   // GBK_TO_UNICODE[19568] := 16#BBEA;
   // GBK_TO_UNICODE[19569] := 16#9B42;
   // GBK_TO_UNICODE[19570] := 16#BBEB;
   // GBK_TO_UNICODE[19571] := 16#6D51;
   // GBK_TO_UNICODE[19572] := 16#BBEC;
   // GBK_TO_UNICODE[19573] := 16#6DF7;
   // GBK_TO_UNICODE[19574] := 16#BBED;
   // GBK_TO_UNICODE[19575] := 16#8C41;
   // GBK_TO_UNICODE[19576] := 16#BBEE;
   // GBK_TO_UNICODE[19577] := 16#6D3B;
   // GBK_TO_UNICODE[19578] := 16#BBEF;
   // GBK_TO_UNICODE[19579] := 16#4F19;
   // GBK_TO_UNICODE[19580] := 16#BBF0;
   // GBK_TO_UNICODE[19581] := 16#706B;
   // GBK_TO_UNICODE[19582] := 16#BBF1;
   // GBK_TO_UNICODE[19583] := 16#83B7;
   // GBK_TO_UNICODE[19584] := 16#BBF2;
   // GBK_TO_UNICODE[19585] := 16#6216;
   // GBK_TO_UNICODE[19586] := 16#BBF3;
   // GBK_TO_UNICODE[19587] := 16#60D1;
   // GBK_TO_UNICODE[19588] := 16#BBF4;
   // GBK_TO_UNICODE[19589] := 16#970D;
   // GBK_TO_UNICODE[19590] := 16#BBF5;
   // GBK_TO_UNICODE[19591] := 16#8D27;
   // GBK_TO_UNICODE[19592] := 16#BBF6;
   // GBK_TO_UNICODE[19593] := 16#7978;
   // GBK_TO_UNICODE[19594] := 16#BBF7;
   // GBK_TO_UNICODE[19595] := 16#51FB;
   // GBK_TO_UNICODE[19596] := 16#BBF8;
   // GBK_TO_UNICODE[19597] := 16#573E;
   // GBK_TO_UNICODE[19598] := 16#BBF9;
   // GBK_TO_UNICODE[19599] := 16#57FA;
   // GBK_TO_UNICODE[19600] := 16#BBFA;
   // GBK_TO_UNICODE[19601] := 16#673A;
   // GBK_TO_UNICODE[19602] := 16#BBFB;
   // GBK_TO_UNICODE[19603] := 16#7578;
   // GBK_TO_UNICODE[19604] := 16#BBFC;
   // GBK_TO_UNICODE[19605] := 16#7A3D;
   // GBK_TO_UNICODE[19606] := 16#BBFD;
   // GBK_TO_UNICODE[19607] := 16#79EF;
   // GBK_TO_UNICODE[19608] := 16#BBFE;
   // GBK_TO_UNICODE[19609] := 16#7B95;
   // GBK_TO_UNICODE[19610] := 16#BC40;
   // GBK_TO_UNICODE[19611] := 16#7CBF;
   // GBK_TO_UNICODE[19612] := 16#BC41;
   // GBK_TO_UNICODE[19613] := 16#7CC0;
   // GBK_TO_UNICODE[19614] := 16#BC42;
   // GBK_TO_UNICODE[19615] := 16#7CC2;
   // GBK_TO_UNICODE[19616] := 16#BC43;
   // GBK_TO_UNICODE[19617] := 16#7CC3;
   // GBK_TO_UNICODE[19618] := 16#BC44;
   // GBK_TO_UNICODE[19619] := 16#7CC4;
   // GBK_TO_UNICODE[19620] := 16#BC45;
   // GBK_TO_UNICODE[19621] := 16#7CC6;
   // GBK_TO_UNICODE[19622] := 16#BC46;
   // GBK_TO_UNICODE[19623] := 16#7CC9;
   // GBK_TO_UNICODE[19624] := 16#BC47;
   // GBK_TO_UNICODE[19625] := 16#7CCB;
   // GBK_TO_UNICODE[19626] := 16#BC48;
   // GBK_TO_UNICODE[19627] := 16#7CCE;
   // GBK_TO_UNICODE[19628] := 16#BC49;
   // GBK_TO_UNICODE[19629] := 16#7CCF;
   // GBK_TO_UNICODE[19630] := 16#BC4A;
   // GBK_TO_UNICODE[19631] := 16#7CD0;
   // GBK_TO_UNICODE[19632] := 16#BC4B;
   // GBK_TO_UNICODE[19633] := 16#7CD1;
   // GBK_TO_UNICODE[19634] := 16#BC4C;
   // GBK_TO_UNICODE[19635] := 16#7CD2;
   // GBK_TO_UNICODE[19636] := 16#BC4D;
   // GBK_TO_UNICODE[19637] := 16#7CD3;
   // GBK_TO_UNICODE[19638] := 16#BC4E;
   // GBK_TO_UNICODE[19639] := 16#7CD4;
   // GBK_TO_UNICODE[19640] := 16#BC4F;
   // GBK_TO_UNICODE[19641] := 16#7CD8;
   // GBK_TO_UNICODE[19642] := 16#BC50;
   // GBK_TO_UNICODE[19643] := 16#7CDA;
   // GBK_TO_UNICODE[19644] := 16#BC51;
   // GBK_TO_UNICODE[19645] := 16#7CDB;
   // GBK_TO_UNICODE[19646] := 16#BC52;
   // GBK_TO_UNICODE[19647] := 16#7CDD;
   // GBK_TO_UNICODE[19648] := 16#BC53;
   // GBK_TO_UNICODE[19649] := 16#7CDE;
   // GBK_TO_UNICODE[19650] := 16#BC54;
   // GBK_TO_UNICODE[19651] := 16#7CE1;
   // GBK_TO_UNICODE[19652] := 16#BC55;
   // GBK_TO_UNICODE[19653] := 16#7CE2;
   // GBK_TO_UNICODE[19654] := 16#BC56;
   // GBK_TO_UNICODE[19655] := 16#7CE3;
   // GBK_TO_UNICODE[19656] := 16#BC57;
   // GBK_TO_UNICODE[19657] := 16#7CE4;
   // GBK_TO_UNICODE[19658] := 16#BC58;
   // GBK_TO_UNICODE[19659] := 16#7CE5;
   // GBK_TO_UNICODE[19660] := 16#BC59;
   // GBK_TO_UNICODE[19661] := 16#7CE6;
   // GBK_TO_UNICODE[19662] := 16#BC5A;
   // GBK_TO_UNICODE[19663] := 16#7CE7;
   // GBK_TO_UNICODE[19664] := 16#BC5B;
   // GBK_TO_UNICODE[19665] := 16#7CE9;
   // GBK_TO_UNICODE[19666] := 16#BC5C;
   // GBK_TO_UNICODE[19667] := 16#7CEA;
   // GBK_TO_UNICODE[19668] := 16#BC5D;
   // GBK_TO_UNICODE[19669] := 16#7CEB;
   // GBK_TO_UNICODE[19670] := 16#BC5E;
   // GBK_TO_UNICODE[19671] := 16#7CEC;
   // GBK_TO_UNICODE[19672] := 16#BC5F;
   // GBK_TO_UNICODE[19673] := 16#7CED;
   // GBK_TO_UNICODE[19674] := 16#BC60;
   // GBK_TO_UNICODE[19675] := 16#7CEE;
   // GBK_TO_UNICODE[19676] := 16#BC61;
   // GBK_TO_UNICODE[19677] := 16#7CF0;
   // GBK_TO_UNICODE[19678] := 16#BC62;
   // GBK_TO_UNICODE[19679] := 16#7CF1;
   // GBK_TO_UNICODE[19680] := 16#BC63;
   // GBK_TO_UNICODE[19681] := 16#7CF2;
   // GBK_TO_UNICODE[19682] := 16#BC64;
   // GBK_TO_UNICODE[19683] := 16#7CF3;
   // GBK_TO_UNICODE[19684] := 16#BC65;
   // GBK_TO_UNICODE[19685] := 16#7CF4;
   // GBK_TO_UNICODE[19686] := 16#BC66;
   // GBK_TO_UNICODE[19687] := 16#7CF5;
   // GBK_TO_UNICODE[19688] := 16#BC67;
   // GBK_TO_UNICODE[19689] := 16#7CF6;
   // GBK_TO_UNICODE[19690] := 16#BC68;
   // GBK_TO_UNICODE[19691] := 16#7CF7;
   // GBK_TO_UNICODE[19692] := 16#BC69;
   // GBK_TO_UNICODE[19693] := 16#7CF9;
   // GBK_TO_UNICODE[19694] := 16#BC6A;
   // GBK_TO_UNICODE[19695] := 16#7CFA;
   // GBK_TO_UNICODE[19696] := 16#BC6B;
   // GBK_TO_UNICODE[19697] := 16#7CFC;
   // GBK_TO_UNICODE[19698] := 16#BC6C;
   // GBK_TO_UNICODE[19699] := 16#7CFD;
   // GBK_TO_UNICODE[19700] := 16#BC6D;
   // GBK_TO_UNICODE[19701] := 16#7CFE;
   // GBK_TO_UNICODE[19702] := 16#BC6E;
   // GBK_TO_UNICODE[19703] := 16#7CFF;
   // GBK_TO_UNICODE[19704] := 16#BC6F;
   // GBK_TO_UNICODE[19705] := 16#7D00;
   // GBK_TO_UNICODE[19706] := 16#BC70;
   // GBK_TO_UNICODE[19707] := 16#7D01;
   // GBK_TO_UNICODE[19708] := 16#BC71;
   // GBK_TO_UNICODE[19709] := 16#7D02;
   // GBK_TO_UNICODE[19710] := 16#BC72;
   // GBK_TO_UNICODE[19711] := 16#7D03;
   // GBK_TO_UNICODE[19712] := 16#BC73;
   // GBK_TO_UNICODE[19713] := 16#7D04;
   // GBK_TO_UNICODE[19714] := 16#BC74;
   // GBK_TO_UNICODE[19715] := 16#7D05;
   // GBK_TO_UNICODE[19716] := 16#BC75;
   // GBK_TO_UNICODE[19717] := 16#7D06;
   // GBK_TO_UNICODE[19718] := 16#BC76;
   // GBK_TO_UNICODE[19719] := 16#7D07;
   // GBK_TO_UNICODE[19720] := 16#BC77;
   // GBK_TO_UNICODE[19721] := 16#7D08;
   // GBK_TO_UNICODE[19722] := 16#BC78;
   // GBK_TO_UNICODE[19723] := 16#7D09;
   // GBK_TO_UNICODE[19724] := 16#BC79;
   // GBK_TO_UNICODE[19725] := 16#7D0B;
   // GBK_TO_UNICODE[19726] := 16#BC7A;
   // GBK_TO_UNICODE[19727] := 16#7D0C;
   // GBK_TO_UNICODE[19728] := 16#BC7B;
   // GBK_TO_UNICODE[19729] := 16#7D0D;
   // GBK_TO_UNICODE[19730] := 16#BC7C;
   // GBK_TO_UNICODE[19731] := 16#7D0E;
   // GBK_TO_UNICODE[19732] := 16#BC7D;
   // GBK_TO_UNICODE[19733] := 16#7D0F;
   // GBK_TO_UNICODE[19734] := 16#BC7E;
   // GBK_TO_UNICODE[19735] := 16#7D10;
   // GBK_TO_UNICODE[19736] := 16#BC80;
   // GBK_TO_UNICODE[19737] := 16#7D11;
   // GBK_TO_UNICODE[19738] := 16#BC81;
   // GBK_TO_UNICODE[19739] := 16#7D12;
   // GBK_TO_UNICODE[19740] := 16#BC82;
   // GBK_TO_UNICODE[19741] := 16#7D13;
   // GBK_TO_UNICODE[19742] := 16#BC83;
   // GBK_TO_UNICODE[19743] := 16#7D14;
   // GBK_TO_UNICODE[19744] := 16#BC84;
   // GBK_TO_UNICODE[19745] := 16#7D15;
   // GBK_TO_UNICODE[19746] := 16#BC85;
   // GBK_TO_UNICODE[19747] := 16#7D16;
   // GBK_TO_UNICODE[19748] := 16#BC86;
   // GBK_TO_UNICODE[19749] := 16#7D17;
   // GBK_TO_UNICODE[19750] := 16#BC87;
   // GBK_TO_UNICODE[19751] := 16#7D18;
   // GBK_TO_UNICODE[19752] := 16#BC88;
   // GBK_TO_UNICODE[19753] := 16#7D19;
   // GBK_TO_UNICODE[19754] := 16#BC89;
   // GBK_TO_UNICODE[19755] := 16#7D1A;
   // GBK_TO_UNICODE[19756] := 16#BC8A;
   // GBK_TO_UNICODE[19757] := 16#7D1B;
   // GBK_TO_UNICODE[19758] := 16#BC8B;
   // GBK_TO_UNICODE[19759] := 16#7D1C;
   // GBK_TO_UNICODE[19760] := 16#BC8C;
   // GBK_TO_UNICODE[19761] := 16#7D1D;
   // GBK_TO_UNICODE[19762] := 16#BC8D;
   // GBK_TO_UNICODE[19763] := 16#7D1E;
   // GBK_TO_UNICODE[19764] := 16#BC8E;
   // GBK_TO_UNICODE[19765] := 16#7D1F;
   // GBK_TO_UNICODE[19766] := 16#BC8F;
   // GBK_TO_UNICODE[19767] := 16#7D21;
   // GBK_TO_UNICODE[19768] := 16#BC90;
   // GBK_TO_UNICODE[19769] := 16#7D23;
   // GBK_TO_UNICODE[19770] := 16#BC91;
   // GBK_TO_UNICODE[19771] := 16#7D24;
   // GBK_TO_UNICODE[19772] := 16#BC92;
   // GBK_TO_UNICODE[19773] := 16#7D25;
   // GBK_TO_UNICODE[19774] := 16#BC93;
   // GBK_TO_UNICODE[19775] := 16#7D26;
   // GBK_TO_UNICODE[19776] := 16#BC94;
   // GBK_TO_UNICODE[19777] := 16#7D28;
   // GBK_TO_UNICODE[19778] := 16#BC95;
   // GBK_TO_UNICODE[19779] := 16#7D29;
   // GBK_TO_UNICODE[19780] := 16#BC96;
   // GBK_TO_UNICODE[19781] := 16#7D2A;
   // GBK_TO_UNICODE[19782] := 16#BC97;
   // GBK_TO_UNICODE[19783] := 16#7D2C;
   // GBK_TO_UNICODE[19784] := 16#BC98;
   // GBK_TO_UNICODE[19785] := 16#7D2D;
   // GBK_TO_UNICODE[19786] := 16#BC99;
   // GBK_TO_UNICODE[19787] := 16#7D2E;
   // GBK_TO_UNICODE[19788] := 16#BC9A;
   // GBK_TO_UNICODE[19789] := 16#7D30;
   // GBK_TO_UNICODE[19790] := 16#BC9B;
   // GBK_TO_UNICODE[19791] := 16#7D31;
   // GBK_TO_UNICODE[19792] := 16#BC9C;
   // GBK_TO_UNICODE[19793] := 16#7D32;
   // GBK_TO_UNICODE[19794] := 16#BC9D;
   // GBK_TO_UNICODE[19795] := 16#7D33;
   // GBK_TO_UNICODE[19796] := 16#BC9E;
   // GBK_TO_UNICODE[19797] := 16#7D34;
   // GBK_TO_UNICODE[19798] := 16#BC9F;
   // GBK_TO_UNICODE[19799] := 16#7D35;
   // GBK_TO_UNICODE[19800] := 16#BCA0;
   // GBK_TO_UNICODE[19801] := 16#7D36;
   // GBK_TO_UNICODE[19802] := 16#BCA1;
   // GBK_TO_UNICODE[19803] := 16#808C;
   // GBK_TO_UNICODE[19804] := 16#BCA2;
   // GBK_TO_UNICODE[19805] := 16#9965;
   // GBK_TO_UNICODE[19806] := 16#BCA3;
   // GBK_TO_UNICODE[19807] := 16#8FF9;
   // GBK_TO_UNICODE[19808] := 16#BCA4;
   // GBK_TO_UNICODE[19809] := 16#6FC0;
   // GBK_TO_UNICODE[19810] := 16#BCA5;
   // GBK_TO_UNICODE[19811] := 16#8BA5;
   // GBK_TO_UNICODE[19812] := 16#BCA6;
   // GBK_TO_UNICODE[19813] := 16#9E21;
   // GBK_TO_UNICODE[19814] := 16#BCA7;
   // GBK_TO_UNICODE[19815] := 16#59EC;
   // GBK_TO_UNICODE[19816] := 16#BCA8;
   // GBK_TO_UNICODE[19817] := 16#7EE9;
   // GBK_TO_UNICODE[19818] := 16#BCA9;
   // GBK_TO_UNICODE[19819] := 16#7F09;
   // GBK_TO_UNICODE[19820] := 16#BCAA;
   // GBK_TO_UNICODE[19821] := 16#5409;
   // GBK_TO_UNICODE[19822] := 16#BCAB;
   // GBK_TO_UNICODE[19823] := 16#6781;
   // GBK_TO_UNICODE[19824] := 16#BCAC;
   // GBK_TO_UNICODE[19825] := 16#68D8;
   // GBK_TO_UNICODE[19826] := 16#BCAD;
   // GBK_TO_UNICODE[19827] := 16#8F91;
   // GBK_TO_UNICODE[19828] := 16#BCAE;
   // GBK_TO_UNICODE[19829] := 16#7C4D;
   // GBK_TO_UNICODE[19830] := 16#BCAF;
   // GBK_TO_UNICODE[19831] := 16#96C6;
   // GBK_TO_UNICODE[19832] := 16#BCB0;
   // GBK_TO_UNICODE[19833] := 16#53CA;
   // GBK_TO_UNICODE[19834] := 16#BCB1;
   // GBK_TO_UNICODE[19835] := 16#6025;
   // GBK_TO_UNICODE[19836] := 16#BCB2;
   // GBK_TO_UNICODE[19837] := 16#75BE;
   // GBK_TO_UNICODE[19838] := 16#BCB3;
   // GBK_TO_UNICODE[19839] := 16#6C72;
   // GBK_TO_UNICODE[19840] := 16#BCB4;
   // GBK_TO_UNICODE[19841] := 16#5373;
   // GBK_TO_UNICODE[19842] := 16#BCB5;
   // GBK_TO_UNICODE[19843] := 16#5AC9;
   // GBK_TO_UNICODE[19844] := 16#BCB6;
   // GBK_TO_UNICODE[19845] := 16#7EA7;
   // GBK_TO_UNICODE[19846] := 16#BCB7;
   // GBK_TO_UNICODE[19847] := 16#6324;
   // GBK_TO_UNICODE[19848] := 16#BCB8;
   // GBK_TO_UNICODE[19849] := 16#51E0;
   // GBK_TO_UNICODE[19850] := 16#BCB9;
   // GBK_TO_UNICODE[19851] := 16#810A;
   // GBK_TO_UNICODE[19852] := 16#BCBA;
   // GBK_TO_UNICODE[19853] := 16#5DF1;
   // GBK_TO_UNICODE[19854] := 16#BCBB;
   // GBK_TO_UNICODE[19855] := 16#84DF;
   // GBK_TO_UNICODE[19856] := 16#BCBC;
   // GBK_TO_UNICODE[19857] := 16#6280;
   // GBK_TO_UNICODE[19858] := 16#BCBD;
   // GBK_TO_UNICODE[19859] := 16#5180;
   // GBK_TO_UNICODE[19860] := 16#BCBE;
   // GBK_TO_UNICODE[19861] := 16#5B63;
   // GBK_TO_UNICODE[19862] := 16#BCBF;
   // GBK_TO_UNICODE[19863] := 16#4F0E;
   // GBK_TO_UNICODE[19864] := 16#BCC0;
   // GBK_TO_UNICODE[19865] := 16#796D;
   // GBK_TO_UNICODE[19866] := 16#BCC1;
   // GBK_TO_UNICODE[19867] := 16#5242;
   // GBK_TO_UNICODE[19868] := 16#BCC2;
   // GBK_TO_UNICODE[19869] := 16#60B8;
   // GBK_TO_UNICODE[19870] := 16#BCC3;
   // GBK_TO_UNICODE[19871] := 16#6D4E;
   // GBK_TO_UNICODE[19872] := 16#BCC4;
   // GBK_TO_UNICODE[19873] := 16#5BC4;
   // GBK_TO_UNICODE[19874] := 16#BCC5;
   // GBK_TO_UNICODE[19875] := 16#5BC2;
   // GBK_TO_UNICODE[19876] := 16#BCC6;
   // GBK_TO_UNICODE[19877] := 16#8BA1;
   // GBK_TO_UNICODE[19878] := 16#BCC7;
   // GBK_TO_UNICODE[19879] := 16#8BB0;
   // GBK_TO_UNICODE[19880] := 16#BCC8;
   // GBK_TO_UNICODE[19881] := 16#65E2;
   // GBK_TO_UNICODE[19882] := 16#BCC9;
   // GBK_TO_UNICODE[19883] := 16#5FCC;
   // GBK_TO_UNICODE[19884] := 16#BCCA;
   // GBK_TO_UNICODE[19885] := 16#9645;
   // GBK_TO_UNICODE[19886] := 16#BCCB;
   // GBK_TO_UNICODE[19887] := 16#5993;
   // GBK_TO_UNICODE[19888] := 16#BCCC;
   // GBK_TO_UNICODE[19889] := 16#7EE7;
   // GBK_TO_UNICODE[19890] := 16#BCCD;
   // GBK_TO_UNICODE[19891] := 16#7EAA;
   // GBK_TO_UNICODE[19892] := 16#BCCE;
   // GBK_TO_UNICODE[19893] := 16#5609;
   // GBK_TO_UNICODE[19894] := 16#BCCF;
   // GBK_TO_UNICODE[19895] := 16#67B7;
   // GBK_TO_UNICODE[19896] := 16#BCD0;
   // GBK_TO_UNICODE[19897] := 16#5939;
   // GBK_TO_UNICODE[19898] := 16#BCD1;
   // GBK_TO_UNICODE[19899] := 16#4F73;
   // GBK_TO_UNICODE[19900] := 16#BCD2;
   // GBK_TO_UNICODE[19901] := 16#5BB6;
   // GBK_TO_UNICODE[19902] := 16#BCD3;
   // GBK_TO_UNICODE[19903] := 16#52A0;
   // GBK_TO_UNICODE[19904] := 16#BCD4;
   // GBK_TO_UNICODE[19905] := 16#835A;
   // GBK_TO_UNICODE[19906] := 16#BCD5;
   // GBK_TO_UNICODE[19907] := 16#988A;
   // GBK_TO_UNICODE[19908] := 16#BCD6;
   // GBK_TO_UNICODE[19909] := 16#8D3E;
   // GBK_TO_UNICODE[19910] := 16#BCD7;
   // GBK_TO_UNICODE[19911] := 16#7532;
   // GBK_TO_UNICODE[19912] := 16#BCD8;
   // GBK_TO_UNICODE[19913] := 16#94BE;
   // GBK_TO_UNICODE[19914] := 16#BCD9;
   // GBK_TO_UNICODE[19915] := 16#5047;
   // GBK_TO_UNICODE[19916] := 16#BCDA;
   // GBK_TO_UNICODE[19917] := 16#7A3C;
   // GBK_TO_UNICODE[19918] := 16#BCDB;
   // GBK_TO_UNICODE[19919] := 16#4EF7;
   // GBK_TO_UNICODE[19920] := 16#BCDC;
   // GBK_TO_UNICODE[19921] := 16#67B6;
   // GBK_TO_UNICODE[19922] := 16#BCDD;
   // GBK_TO_UNICODE[19923] := 16#9A7E;
   // GBK_TO_UNICODE[19924] := 16#BCDE;
   // GBK_TO_UNICODE[19925] := 16#5AC1;
   // GBK_TO_UNICODE[19926] := 16#BCDF;
   // GBK_TO_UNICODE[19927] := 16#6B7C;
   // GBK_TO_UNICODE[19928] := 16#BCE0;
   // GBK_TO_UNICODE[19929] := 16#76D1;
   // GBK_TO_UNICODE[19930] := 16#BCE1;
   // GBK_TO_UNICODE[19931] := 16#575A;
   // GBK_TO_UNICODE[19932] := 16#BCE2;
   // GBK_TO_UNICODE[19933] := 16#5C16;
   // GBK_TO_UNICODE[19934] := 16#BCE3;
   // GBK_TO_UNICODE[19935] := 16#7B3A;
   // GBK_TO_UNICODE[19936] := 16#BCE4;
   // GBK_TO_UNICODE[19937] := 16#95F4;
   // GBK_TO_UNICODE[19938] := 16#BCE5;
   // GBK_TO_UNICODE[19939] := 16#714E;
   // GBK_TO_UNICODE[19940] := 16#BCE6;
   // GBK_TO_UNICODE[19941] := 16#517C;
   // GBK_TO_UNICODE[19942] := 16#BCE7;
   // GBK_TO_UNICODE[19943] := 16#80A9;
   // GBK_TO_UNICODE[19944] := 16#BCE8;
   // GBK_TO_UNICODE[19945] := 16#8270;
   // GBK_TO_UNICODE[19946] := 16#BCE9;
   // GBK_TO_UNICODE[19947] := 16#5978;
   // GBK_TO_UNICODE[19948] := 16#BCEA;
   // GBK_TO_UNICODE[19949] := 16#7F04;
   // GBK_TO_UNICODE[19950] := 16#BCEB;
   // GBK_TO_UNICODE[19951] := 16#8327;
   // GBK_TO_UNICODE[19952] := 16#BCEC;
   // GBK_TO_UNICODE[19953] := 16#68C0;
   // GBK_TO_UNICODE[19954] := 16#BCED;
   // GBK_TO_UNICODE[19955] := 16#67EC;
   // GBK_TO_UNICODE[19956] := 16#BCEE;
   // GBK_TO_UNICODE[19957] := 16#78B1;
   // GBK_TO_UNICODE[19958] := 16#BCEF;
   // GBK_TO_UNICODE[19959] := 16#7877;
   // GBK_TO_UNICODE[19960] := 16#BCF0;
   // GBK_TO_UNICODE[19961] := 16#62E3;
   // GBK_TO_UNICODE[19962] := 16#BCF1;
   // GBK_TO_UNICODE[19963] := 16#6361;
   // GBK_TO_UNICODE[19964] := 16#BCF2;
   // GBK_TO_UNICODE[19965] := 16#7B80;
   // GBK_TO_UNICODE[19966] := 16#BCF3;
   // GBK_TO_UNICODE[19967] := 16#4FED;
   // GBK_TO_UNICODE[19968] := 16#BCF4;
   // GBK_TO_UNICODE[19969] := 16#526A;
   // GBK_TO_UNICODE[19970] := 16#BCF5;
   // GBK_TO_UNICODE[19971] := 16#51CF;
   // GBK_TO_UNICODE[19972] := 16#BCF6;
   // GBK_TO_UNICODE[19973] := 16#8350;
   // GBK_TO_UNICODE[19974] := 16#BCF7;
   // GBK_TO_UNICODE[19975] := 16#69DB;
   // GBK_TO_UNICODE[19976] := 16#BCF8;
   // GBK_TO_UNICODE[19977] := 16#9274;
   // GBK_TO_UNICODE[19978] := 16#BCF9;
   // GBK_TO_UNICODE[19979] := 16#8DF5;
   // GBK_TO_UNICODE[19980] := 16#BCFA;
   // GBK_TO_UNICODE[19981] := 16#8D31;
   // GBK_TO_UNICODE[19982] := 16#BCFB;
   // GBK_TO_UNICODE[19983] := 16#89C1;
   // GBK_TO_UNICODE[19984] := 16#BCFC;
   // GBK_TO_UNICODE[19985] := 16#952E;
   // GBK_TO_UNICODE[19986] := 16#BCFD;
   // GBK_TO_UNICODE[19987] := 16#7BAD;
   // GBK_TO_UNICODE[19988] := 16#BCFE;
   // GBK_TO_UNICODE[19989] := 16#4EF6;
   // GBK_TO_UNICODE[19990] := 16#BD40;
   // GBK_TO_UNICODE[19991] := 16#7D37;
   // GBK_TO_UNICODE[19992] := 16#BD41;
   // GBK_TO_UNICODE[19993] := 16#7D38;
   // GBK_TO_UNICODE[19994] := 16#BD42;
   // GBK_TO_UNICODE[19995] := 16#7D39;
   // GBK_TO_UNICODE[19996] := 16#BD43;
   // GBK_TO_UNICODE[19997] := 16#7D3A;
   // GBK_TO_UNICODE[19998] := 16#BD44;
   // GBK_TO_UNICODE[19999] := 16#7D3B;
   // GBK_TO_UNICODE[20000] := 16#BD45;
   // GBK_TO_UNICODE[20001] := 16#7D3C;
   // GBK_TO_UNICODE[20002] := 16#BD46;
   // GBK_TO_UNICODE[20003] := 16#7D3D;
   // GBK_TO_UNICODE[20004] := 16#BD47;
   // GBK_TO_UNICODE[20005] := 16#7D3E;
   // GBK_TO_UNICODE[20006] := 16#BD48;
   // GBK_TO_UNICODE[20007] := 16#7D3F;
   // GBK_TO_UNICODE[20008] := 16#BD49;
   // GBK_TO_UNICODE[20009] := 16#7D40;
   // GBK_TO_UNICODE[20010] := 16#BD4A;
   // GBK_TO_UNICODE[20011] := 16#7D41;
   // GBK_TO_UNICODE[20012] := 16#BD4B;
   // GBK_TO_UNICODE[20013] := 16#7D42;
   // GBK_TO_UNICODE[20014] := 16#BD4C;
   // GBK_TO_UNICODE[20015] := 16#7D43;
   // GBK_TO_UNICODE[20016] := 16#BD4D;
   // GBK_TO_UNICODE[20017] := 16#7D44;
   // GBK_TO_UNICODE[20018] := 16#BD4E;
   // GBK_TO_UNICODE[20019] := 16#7D45;
   // GBK_TO_UNICODE[20020] := 16#BD4F;
   // GBK_TO_UNICODE[20021] := 16#7D46;
   // GBK_TO_UNICODE[20022] := 16#BD50;
   // GBK_TO_UNICODE[20023] := 16#7D47;
   // GBK_TO_UNICODE[20024] := 16#BD51;
   // GBK_TO_UNICODE[20025] := 16#7D48;
   // GBK_TO_UNICODE[20026] := 16#BD52;
   // GBK_TO_UNICODE[20027] := 16#7D49;
   // GBK_TO_UNICODE[20028] := 16#BD53;
   // GBK_TO_UNICODE[20029] := 16#7D4A;
   // GBK_TO_UNICODE[20030] := 16#BD54;
   // GBK_TO_UNICODE[20031] := 16#7D4B;
   // GBK_TO_UNICODE[20032] := 16#BD55;
   // GBK_TO_UNICODE[20033] := 16#7D4C;
   // GBK_TO_UNICODE[20034] := 16#BD56;
   // GBK_TO_UNICODE[20035] := 16#7D4D;
   // GBK_TO_UNICODE[20036] := 16#BD57;
   // GBK_TO_UNICODE[20037] := 16#7D4E;
   // GBK_TO_UNICODE[20038] := 16#BD58;
   // GBK_TO_UNICODE[20039] := 16#7D4F;
   // GBK_TO_UNICODE[20040] := 16#BD59;
   // GBK_TO_UNICODE[20041] := 16#7D50;
   // GBK_TO_UNICODE[20042] := 16#BD5A;
   // GBK_TO_UNICODE[20043] := 16#7D51;
   // GBK_TO_UNICODE[20044] := 16#BD5B;
   // GBK_TO_UNICODE[20045] := 16#7D52;
   // GBK_TO_UNICODE[20046] := 16#BD5C;
   // GBK_TO_UNICODE[20047] := 16#7D53;
   // GBK_TO_UNICODE[20048] := 16#BD5D;
   // GBK_TO_UNICODE[20049] := 16#7D54;
   // GBK_TO_UNICODE[20050] := 16#BD5E;
   // GBK_TO_UNICODE[20051] := 16#7D55;
   // GBK_TO_UNICODE[20052] := 16#BD5F;
   // GBK_TO_UNICODE[20053] := 16#7D56;
   // GBK_TO_UNICODE[20054] := 16#BD60;
   // GBK_TO_UNICODE[20055] := 16#7D57;
   // GBK_TO_UNICODE[20056] := 16#BD61;
   // GBK_TO_UNICODE[20057] := 16#7D58;
   // GBK_TO_UNICODE[20058] := 16#BD62;
   // GBK_TO_UNICODE[20059] := 16#7D59;
   // GBK_TO_UNICODE[20060] := 16#BD63;
   // GBK_TO_UNICODE[20061] := 16#7D5A;
   // GBK_TO_UNICODE[20062] := 16#BD64;
   // GBK_TO_UNICODE[20063] := 16#7D5B;
   // GBK_TO_UNICODE[20064] := 16#BD65;
   // GBK_TO_UNICODE[20065] := 16#7D5C;
   // GBK_TO_UNICODE[20066] := 16#BD66;
   // GBK_TO_UNICODE[20067] := 16#7D5D;
   // GBK_TO_UNICODE[20068] := 16#BD67;
   // GBK_TO_UNICODE[20069] := 16#7D5E;
   // GBK_TO_UNICODE[20070] := 16#BD68;
   // GBK_TO_UNICODE[20071] := 16#7D5F;
   // GBK_TO_UNICODE[20072] := 16#BD69;
   // GBK_TO_UNICODE[20073] := 16#7D60;
   // GBK_TO_UNICODE[20074] := 16#BD6A;
   // GBK_TO_UNICODE[20075] := 16#7D61;
   // GBK_TO_UNICODE[20076] := 16#BD6B;
   // GBK_TO_UNICODE[20077] := 16#7D62;
   // GBK_TO_UNICODE[20078] := 16#BD6C;
   // GBK_TO_UNICODE[20079] := 16#7D63;
   // GBK_TO_UNICODE[20080] := 16#BD6D;
   // GBK_TO_UNICODE[20081] := 16#7D64;
   // GBK_TO_UNICODE[20082] := 16#BD6E;
   // GBK_TO_UNICODE[20083] := 16#7D65;
   // GBK_TO_UNICODE[20084] := 16#BD6F;
   // GBK_TO_UNICODE[20085] := 16#7D66;
   // GBK_TO_UNICODE[20086] := 16#BD70;
   // GBK_TO_UNICODE[20087] := 16#7D67;
   // GBK_TO_UNICODE[20088] := 16#BD71;
   // GBK_TO_UNICODE[20089] := 16#7D68;
   // GBK_TO_UNICODE[20090] := 16#BD72;
   // GBK_TO_UNICODE[20091] := 16#7D69;
   // GBK_TO_UNICODE[20092] := 16#BD73;
   // GBK_TO_UNICODE[20093] := 16#7D6A;
   // GBK_TO_UNICODE[20094] := 16#BD74;
   // GBK_TO_UNICODE[20095] := 16#7D6B;
   // GBK_TO_UNICODE[20096] := 16#BD75;
   // GBK_TO_UNICODE[20097] := 16#7D6C;
   // GBK_TO_UNICODE[20098] := 16#BD76;
   // GBK_TO_UNICODE[20099] := 16#7D6D;
   // GBK_TO_UNICODE[20100] := 16#BD77;
   // GBK_TO_UNICODE[20101] := 16#7D6F;
   // GBK_TO_UNICODE[20102] := 16#BD78;
   // GBK_TO_UNICODE[20103] := 16#7D70;
   // GBK_TO_UNICODE[20104] := 16#BD79;
   // GBK_TO_UNICODE[20105] := 16#7D71;
   // GBK_TO_UNICODE[20106] := 16#BD7A;
   // GBK_TO_UNICODE[20107] := 16#7D72;
   // GBK_TO_UNICODE[20108] := 16#BD7B;
   // GBK_TO_UNICODE[20109] := 16#7D73;
   // GBK_TO_UNICODE[20110] := 16#BD7C;
   // GBK_TO_UNICODE[20111] := 16#7D74;
   // GBK_TO_UNICODE[20112] := 16#BD7D;
   // GBK_TO_UNICODE[20113] := 16#7D75;
   // GBK_TO_UNICODE[20114] := 16#BD7E;
   // GBK_TO_UNICODE[20115] := 16#7D76;
   // GBK_TO_UNICODE[20116] := 16#BD80;
   // GBK_TO_UNICODE[20117] := 16#7D78;
   // GBK_TO_UNICODE[20118] := 16#BD81;
   // GBK_TO_UNICODE[20119] := 16#7D79;
   // GBK_TO_UNICODE[20120] := 16#BD82;
   // GBK_TO_UNICODE[20121] := 16#7D7A;
   // GBK_TO_UNICODE[20122] := 16#BD83;
   // GBK_TO_UNICODE[20123] := 16#7D7B;
   // GBK_TO_UNICODE[20124] := 16#BD84;
   // GBK_TO_UNICODE[20125] := 16#7D7C;
   // GBK_TO_UNICODE[20126] := 16#BD85;
   // GBK_TO_UNICODE[20127] := 16#7D7D;
   // GBK_TO_UNICODE[20128] := 16#BD86;
   // GBK_TO_UNICODE[20129] := 16#7D7E;
   // GBK_TO_UNICODE[20130] := 16#BD87;
   // GBK_TO_UNICODE[20131] := 16#7D7F;
   // GBK_TO_UNICODE[20132] := 16#BD88;
   // GBK_TO_UNICODE[20133] := 16#7D80;
   // GBK_TO_UNICODE[20134] := 16#BD89;
   // GBK_TO_UNICODE[20135] := 16#7D81;
   // GBK_TO_UNICODE[20136] := 16#BD8A;
   // GBK_TO_UNICODE[20137] := 16#7D82;
   // GBK_TO_UNICODE[20138] := 16#BD8B;
   // GBK_TO_UNICODE[20139] := 16#7D83;
   // GBK_TO_UNICODE[20140] := 16#BD8C;
   // GBK_TO_UNICODE[20141] := 16#7D84;
   // GBK_TO_UNICODE[20142] := 16#BD8D;
   // GBK_TO_UNICODE[20143] := 16#7D85;
   // GBK_TO_UNICODE[20144] := 16#BD8E;
   // GBK_TO_UNICODE[20145] := 16#7D86;
   // GBK_TO_UNICODE[20146] := 16#BD8F;
   // GBK_TO_UNICODE[20147] := 16#7D87;
   // GBK_TO_UNICODE[20148] := 16#BD90;
   // GBK_TO_UNICODE[20149] := 16#7D88;
   // GBK_TO_UNICODE[20150] := 16#BD91;
   // GBK_TO_UNICODE[20151] := 16#7D89;
   // GBK_TO_UNICODE[20152] := 16#BD92;
   // GBK_TO_UNICODE[20153] := 16#7D8A;
   // GBK_TO_UNICODE[20154] := 16#BD93;
   // GBK_TO_UNICODE[20155] := 16#7D8B;
   // GBK_TO_UNICODE[20156] := 16#BD94;
   // GBK_TO_UNICODE[20157] := 16#7D8C;
   // GBK_TO_UNICODE[20158] := 16#BD95;
   // GBK_TO_UNICODE[20159] := 16#7D8D;
   // GBK_TO_UNICODE[20160] := 16#BD96;
   // GBK_TO_UNICODE[20161] := 16#7D8E;
   // GBK_TO_UNICODE[20162] := 16#BD97;
   // GBK_TO_UNICODE[20163] := 16#7D8F;
   // GBK_TO_UNICODE[20164] := 16#BD98;
   // GBK_TO_UNICODE[20165] := 16#7D90;
   // GBK_TO_UNICODE[20166] := 16#BD99;
   // GBK_TO_UNICODE[20167] := 16#7D91;
   // GBK_TO_UNICODE[20168] := 16#BD9A;
   // GBK_TO_UNICODE[20169] := 16#7D92;
   // GBK_TO_UNICODE[20170] := 16#BD9B;
   // GBK_TO_UNICODE[20171] := 16#7D93;
   // GBK_TO_UNICODE[20172] := 16#BD9C;
   // GBK_TO_UNICODE[20173] := 16#7D94;
   // GBK_TO_UNICODE[20174] := 16#BD9D;
   // GBK_TO_UNICODE[20175] := 16#7D95;
   // GBK_TO_UNICODE[20176] := 16#BD9E;
   // GBK_TO_UNICODE[20177] := 16#7D96;
   // GBK_TO_UNICODE[20178] := 16#BD9F;
   // GBK_TO_UNICODE[20179] := 16#7D97;
   // GBK_TO_UNICODE[20180] := 16#BDA0;
   // GBK_TO_UNICODE[20181] := 16#7D98;
   // GBK_TO_UNICODE[20182] := 16#BDA1;
   // GBK_TO_UNICODE[20183] := 16#5065;
   // GBK_TO_UNICODE[20184] := 16#BDA2;
   // GBK_TO_UNICODE[20185] := 16#8230;
   // GBK_TO_UNICODE[20186] := 16#BDA3;
   // GBK_TO_UNICODE[20187] := 16#5251;
   // GBK_TO_UNICODE[20188] := 16#BDA4;
   // GBK_TO_UNICODE[20189] := 16#996F;
   // GBK_TO_UNICODE[20190] := 16#BDA5;
   // GBK_TO_UNICODE[20191] := 16#6E10;
   // GBK_TO_UNICODE[20192] := 16#BDA6;
   // GBK_TO_UNICODE[20193] := 16#6E85;
   // GBK_TO_UNICODE[20194] := 16#BDA7;
   // GBK_TO_UNICODE[20195] := 16#6DA7;
   // GBK_TO_UNICODE[20196] := 16#BDA8;
   // GBK_TO_UNICODE[20197] := 16#5EFA;
   // GBK_TO_UNICODE[20198] := 16#BDA9;
   // GBK_TO_UNICODE[20199] := 16#50F5;
   // GBK_TO_UNICODE[20200] := 16#BDAA;
   // GBK_TO_UNICODE[20201] := 16#59DC;
   // GBK_TO_UNICODE[20202] := 16#BDAB;
   // GBK_TO_UNICODE[20203] := 16#5C06;
   // GBK_TO_UNICODE[20204] := 16#BDAC;
   // GBK_TO_UNICODE[20205] := 16#6D46;
   // GBK_TO_UNICODE[20206] := 16#BDAD;
   // GBK_TO_UNICODE[20207] := 16#6C5F;
   // GBK_TO_UNICODE[20208] := 16#BDAE;
   // GBK_TO_UNICODE[20209] := 16#7586;
   // GBK_TO_UNICODE[20210] := 16#BDAF;
   // GBK_TO_UNICODE[20211] := 16#848B;
   // GBK_TO_UNICODE[20212] := 16#BDB0;
   // GBK_TO_UNICODE[20213] := 16#6868;
   // GBK_TO_UNICODE[20214] := 16#BDB1;
   // GBK_TO_UNICODE[20215] := 16#5956;
   // GBK_TO_UNICODE[20216] := 16#BDB2;
   // GBK_TO_UNICODE[20217] := 16#8BB2;
   // GBK_TO_UNICODE[20218] := 16#BDB3;
   // GBK_TO_UNICODE[20219] := 16#5320;
   // GBK_TO_UNICODE[20220] := 16#BDB4;
   // GBK_TO_UNICODE[20221] := 16#9171;
   // GBK_TO_UNICODE[20222] := 16#BDB5;
   // GBK_TO_UNICODE[20223] := 16#964D;
   // GBK_TO_UNICODE[20224] := 16#BDB6;
   // GBK_TO_UNICODE[20225] := 16#8549;
   // GBK_TO_UNICODE[20226] := 16#BDB7;
   // GBK_TO_UNICODE[20227] := 16#6912;
   // GBK_TO_UNICODE[20228] := 16#BDB8;
   // GBK_TO_UNICODE[20229] := 16#7901;
   // GBK_TO_UNICODE[20230] := 16#BDB9;
   // GBK_TO_UNICODE[20231] := 16#7126;
   // GBK_TO_UNICODE[20232] := 16#BDBA;
   // GBK_TO_UNICODE[20233] := 16#80F6;
   // GBK_TO_UNICODE[20234] := 16#BDBB;
   // GBK_TO_UNICODE[20235] := 16#4EA4;
   // GBK_TO_UNICODE[20236] := 16#BDBC;
   // GBK_TO_UNICODE[20237] := 16#90CA;
   // GBK_TO_UNICODE[20238] := 16#BDBD;
   // GBK_TO_UNICODE[20239] := 16#6D47;
   // GBK_TO_UNICODE[20240] := 16#BDBE;
   // GBK_TO_UNICODE[20241] := 16#9A84;
   // GBK_TO_UNICODE[20242] := 16#BDBF;
   // GBK_TO_UNICODE[20243] := 16#5A07;
   // GBK_TO_UNICODE[20244] := 16#BDC0;
   // GBK_TO_UNICODE[20245] := 16#56BC;
   // GBK_TO_UNICODE[20246] := 16#BDC1;
   // GBK_TO_UNICODE[20247] := 16#6405;
   // GBK_TO_UNICODE[20248] := 16#BDC2;
   // GBK_TO_UNICODE[20249] := 16#94F0;
   // GBK_TO_UNICODE[20250] := 16#BDC3;
   // GBK_TO_UNICODE[20251] := 16#77EB;
   // GBK_TO_UNICODE[20252] := 16#BDC4;
   // GBK_TO_UNICODE[20253] := 16#4FA5;
   // GBK_TO_UNICODE[20254] := 16#BDC5;
   // GBK_TO_UNICODE[20255] := 16#811A;
   // GBK_TO_UNICODE[20256] := 16#BDC6;
   // GBK_TO_UNICODE[20257] := 16#72E1;
   // GBK_TO_UNICODE[20258] := 16#BDC7;
   // GBK_TO_UNICODE[20259] := 16#89D2;
   // GBK_TO_UNICODE[20260] := 16#BDC8;
   // GBK_TO_UNICODE[20261] := 16#997A;
   // GBK_TO_UNICODE[20262] := 16#BDC9;
   // GBK_TO_UNICODE[20263] := 16#7F34;
   // GBK_TO_UNICODE[20264] := 16#BDCA;
   // GBK_TO_UNICODE[20265] := 16#7EDE;
   // GBK_TO_UNICODE[20266] := 16#BDCB;
   // GBK_TO_UNICODE[20267] := 16#527F;
   // GBK_TO_UNICODE[20268] := 16#BDCC;
   // GBK_TO_UNICODE[20269] := 16#6559;
   // GBK_TO_UNICODE[20270] := 16#BDCD;
   // GBK_TO_UNICODE[20271] := 16#9175;
   // GBK_TO_UNICODE[20272] := 16#BDCE;
   // GBK_TO_UNICODE[20273] := 16#8F7F;
   // GBK_TO_UNICODE[20274] := 16#BDCF;
   // GBK_TO_UNICODE[20275] := 16#8F83;
   // GBK_TO_UNICODE[20276] := 16#BDD0;
   // GBK_TO_UNICODE[20277] := 16#53EB;
   // GBK_TO_UNICODE[20278] := 16#BDD1;
   // GBK_TO_UNICODE[20279] := 16#7A96;
   // GBK_TO_UNICODE[20280] := 16#BDD2;
   // GBK_TO_UNICODE[20281] := 16#63ED;
   // GBK_TO_UNICODE[20282] := 16#BDD3;
   // GBK_TO_UNICODE[20283] := 16#63A5;
   // GBK_TO_UNICODE[20284] := 16#BDD4;
   // GBK_TO_UNICODE[20285] := 16#7686;
   // GBK_TO_UNICODE[20286] := 16#BDD5;
   // GBK_TO_UNICODE[20287] := 16#79F8;
   // GBK_TO_UNICODE[20288] := 16#BDD6;
   // GBK_TO_UNICODE[20289] := 16#8857;
   // GBK_TO_UNICODE[20290] := 16#BDD7;
   // GBK_TO_UNICODE[20291] := 16#9636;
   // GBK_TO_UNICODE[20292] := 16#BDD8;
   // GBK_TO_UNICODE[20293] := 16#622A;
   // GBK_TO_UNICODE[20294] := 16#BDD9;
   // GBK_TO_UNICODE[20295] := 16#52AB;
   // GBK_TO_UNICODE[20296] := 16#BDDA;
   // GBK_TO_UNICODE[20297] := 16#8282;
   // GBK_TO_UNICODE[20298] := 16#BDDB;
   // GBK_TO_UNICODE[20299] := 16#6854;
   // GBK_TO_UNICODE[20300] := 16#BDDC;
   // GBK_TO_UNICODE[20301] := 16#6770;
   // GBK_TO_UNICODE[20302] := 16#BDDD;
   // GBK_TO_UNICODE[20303] := 16#6377;
   // GBK_TO_UNICODE[20304] := 16#BDDE;
   // GBK_TO_UNICODE[20305] := 16#776B;
   // GBK_TO_UNICODE[20306] := 16#BDDF;
   // GBK_TO_UNICODE[20307] := 16#7AED;
   // GBK_TO_UNICODE[20308] := 16#BDE0;
   // GBK_TO_UNICODE[20309] := 16#6D01;
   // GBK_TO_UNICODE[20310] := 16#BDE1;
   // GBK_TO_UNICODE[20311] := 16#7ED3;
   // GBK_TO_UNICODE[20312] := 16#BDE2;
   // GBK_TO_UNICODE[20313] := 16#89E3;
   // GBK_TO_UNICODE[20314] := 16#BDE3;
   // GBK_TO_UNICODE[20315] := 16#59D0;
   // GBK_TO_UNICODE[20316] := 16#BDE4;
   // GBK_TO_UNICODE[20317] := 16#6212;
   // GBK_TO_UNICODE[20318] := 16#BDE5;
   // GBK_TO_UNICODE[20319] := 16#85C9;
   // GBK_TO_UNICODE[20320] := 16#BDE6;
   // GBK_TO_UNICODE[20321] := 16#82A5;
   // GBK_TO_UNICODE[20322] := 16#BDE7;
   // GBK_TO_UNICODE[20323] := 16#754C;
   // GBK_TO_UNICODE[20324] := 16#BDE8;
   // GBK_TO_UNICODE[20325] := 16#501F;
   // GBK_TO_UNICODE[20326] := 16#BDE9;
   // GBK_TO_UNICODE[20327] := 16#4ECB;
   // GBK_TO_UNICODE[20328] := 16#BDEA;
   // GBK_TO_UNICODE[20329] := 16#75A5;
   // GBK_TO_UNICODE[20330] := 16#BDEB;
   // GBK_TO_UNICODE[20331] := 16#8BEB;
   // GBK_TO_UNICODE[20332] := 16#BDEC;
   // GBK_TO_UNICODE[20333] := 16#5C4A;
   // GBK_TO_UNICODE[20334] := 16#BDED;
   // GBK_TO_UNICODE[20335] := 16#5DFE;
   // GBK_TO_UNICODE[20336] := 16#BDEE;
   // GBK_TO_UNICODE[20337] := 16#7B4B;
   // GBK_TO_UNICODE[20338] := 16#BDEF;
   // GBK_TO_UNICODE[20339] := 16#65A4;
   // GBK_TO_UNICODE[20340] := 16#BDF0;
   // GBK_TO_UNICODE[20341] := 16#91D1;
   // GBK_TO_UNICODE[20342] := 16#BDF1;
   // GBK_TO_UNICODE[20343] := 16#4ECA;
   // GBK_TO_UNICODE[20344] := 16#BDF2;
   // GBK_TO_UNICODE[20345] := 16#6D25;
   // GBK_TO_UNICODE[20346] := 16#BDF3;
   // GBK_TO_UNICODE[20347] := 16#895F;
   // GBK_TO_UNICODE[20348] := 16#BDF4;
   // GBK_TO_UNICODE[20349] := 16#7D27;
   // GBK_TO_UNICODE[20350] := 16#BDF5;
   // GBK_TO_UNICODE[20351] := 16#9526;
   // GBK_TO_UNICODE[20352] := 16#BDF6;
   // GBK_TO_UNICODE[20353] := 16#4EC5;
   // GBK_TO_UNICODE[20354] := 16#BDF7;
   // GBK_TO_UNICODE[20355] := 16#8C28;
   // GBK_TO_UNICODE[20356] := 16#BDF8;
   // GBK_TO_UNICODE[20357] := 16#8FDB;
   // GBK_TO_UNICODE[20358] := 16#BDF9;
   // GBK_TO_UNICODE[20359] := 16#9773;
   // GBK_TO_UNICODE[20360] := 16#BDFA;
   // GBK_TO_UNICODE[20361] := 16#664B;
   // GBK_TO_UNICODE[20362] := 16#BDFB;
   // GBK_TO_UNICODE[20363] := 16#7981;
   // GBK_TO_UNICODE[20364] := 16#BDFC;
   // GBK_TO_UNICODE[20365] := 16#8FD1;
   // GBK_TO_UNICODE[20366] := 16#BDFD;
   // GBK_TO_UNICODE[20367] := 16#70EC;
   // GBK_TO_UNICODE[20368] := 16#BDFE;
   // GBK_TO_UNICODE[20369] := 16#6D78;
   // GBK_TO_UNICODE[20370] := 16#BE40;
   // GBK_TO_UNICODE[20371] := 16#7D99;
   // GBK_TO_UNICODE[20372] := 16#BE41;
   // GBK_TO_UNICODE[20373] := 16#7D9A;
   // GBK_TO_UNICODE[20374] := 16#BE42;
   // GBK_TO_UNICODE[20375] := 16#7D9B;
   // GBK_TO_UNICODE[20376] := 16#BE43;
   // GBK_TO_UNICODE[20377] := 16#7D9C;
   // GBK_TO_UNICODE[20378] := 16#BE44;
   // GBK_TO_UNICODE[20379] := 16#7D9D;
   // GBK_TO_UNICODE[20380] := 16#BE45;
   // GBK_TO_UNICODE[20381] := 16#7D9E;
   // GBK_TO_UNICODE[20382] := 16#BE46;
   // GBK_TO_UNICODE[20383] := 16#7D9F;
   // GBK_TO_UNICODE[20384] := 16#BE47;
   // GBK_TO_UNICODE[20385] := 16#7DA0;
   // GBK_TO_UNICODE[20386] := 16#BE48;
   // GBK_TO_UNICODE[20387] := 16#7DA1;
   // GBK_TO_UNICODE[20388] := 16#BE49;
   // GBK_TO_UNICODE[20389] := 16#7DA2;
   // GBK_TO_UNICODE[20390] := 16#BE4A;
   // GBK_TO_UNICODE[20391] := 16#7DA3;
   // GBK_TO_UNICODE[20392] := 16#BE4B;
   // GBK_TO_UNICODE[20393] := 16#7DA4;
   // GBK_TO_UNICODE[20394] := 16#BE4C;
   // GBK_TO_UNICODE[20395] := 16#7DA5;
   // GBK_TO_UNICODE[20396] := 16#BE4D;
   // GBK_TO_UNICODE[20397] := 16#7DA7;
   // GBK_TO_UNICODE[20398] := 16#BE4E;
   // GBK_TO_UNICODE[20399] := 16#7DA8;
   // GBK_TO_UNICODE[20400] := 16#BE4F;
   // GBK_TO_UNICODE[20401] := 16#7DA9;
   // GBK_TO_UNICODE[20402] := 16#BE50;
   // GBK_TO_UNICODE[20403] := 16#7DAA;
   // GBK_TO_UNICODE[20404] := 16#BE51;
   // GBK_TO_UNICODE[20405] := 16#7DAB;
   // GBK_TO_UNICODE[20406] := 16#BE52;
   // GBK_TO_UNICODE[20407] := 16#7DAC;
   // GBK_TO_UNICODE[20408] := 16#BE53;
   // GBK_TO_UNICODE[20409] := 16#7DAD;
   // GBK_TO_UNICODE[20410] := 16#BE54;
   // GBK_TO_UNICODE[20411] := 16#7DAF;
   // GBK_TO_UNICODE[20412] := 16#BE55;
   // GBK_TO_UNICODE[20413] := 16#7DB0;
   // GBK_TO_UNICODE[20414] := 16#BE56;
   // GBK_TO_UNICODE[20415] := 16#7DB1;
   // GBK_TO_UNICODE[20416] := 16#BE57;
   // GBK_TO_UNICODE[20417] := 16#7DB2;
   // GBK_TO_UNICODE[20418] := 16#BE58;
   // GBK_TO_UNICODE[20419] := 16#7DB3;
   // GBK_TO_UNICODE[20420] := 16#BE59;
   // GBK_TO_UNICODE[20421] := 16#7DB4;
   // GBK_TO_UNICODE[20422] := 16#BE5A;
   // GBK_TO_UNICODE[20423] := 16#7DB5;
   // GBK_TO_UNICODE[20424] := 16#BE5B;
   // GBK_TO_UNICODE[20425] := 16#7DB6;
   // GBK_TO_UNICODE[20426] := 16#BE5C;
   // GBK_TO_UNICODE[20427] := 16#7DB7;
   // GBK_TO_UNICODE[20428] := 16#BE5D;
   // GBK_TO_UNICODE[20429] := 16#7DB8;
   // GBK_TO_UNICODE[20430] := 16#BE5E;
   // GBK_TO_UNICODE[20431] := 16#7DB9;
   // GBK_TO_UNICODE[20432] := 16#BE5F;
   // GBK_TO_UNICODE[20433] := 16#7DBA;
   // GBK_TO_UNICODE[20434] := 16#BE60;
   // GBK_TO_UNICODE[20435] := 16#7DBB;
   // GBK_TO_UNICODE[20436] := 16#BE61;
   // GBK_TO_UNICODE[20437] := 16#7DBC;
   // GBK_TO_UNICODE[20438] := 16#BE62;
   // GBK_TO_UNICODE[20439] := 16#7DBD;
   // GBK_TO_UNICODE[20440] := 16#BE63;
   // GBK_TO_UNICODE[20441] := 16#7DBE;
   // GBK_TO_UNICODE[20442] := 16#BE64;
   // GBK_TO_UNICODE[20443] := 16#7DBF;
   // GBK_TO_UNICODE[20444] := 16#BE65;
   // GBK_TO_UNICODE[20445] := 16#7DC0;
   // GBK_TO_UNICODE[20446] := 16#BE66;
   // GBK_TO_UNICODE[20447] := 16#7DC1;
   // GBK_TO_UNICODE[20448] := 16#BE67;
   // GBK_TO_UNICODE[20449] := 16#7DC2;
   // GBK_TO_UNICODE[20450] := 16#BE68;
   // GBK_TO_UNICODE[20451] := 16#7DC3;
   // GBK_TO_UNICODE[20452] := 16#BE69;
   // GBK_TO_UNICODE[20453] := 16#7DC4;
   // GBK_TO_UNICODE[20454] := 16#BE6A;
   // GBK_TO_UNICODE[20455] := 16#7DC5;
   // GBK_TO_UNICODE[20456] := 16#BE6B;
   // GBK_TO_UNICODE[20457] := 16#7DC6;
   // GBK_TO_UNICODE[20458] := 16#BE6C;
   // GBK_TO_UNICODE[20459] := 16#7DC7;
   // GBK_TO_UNICODE[20460] := 16#BE6D;
   // GBK_TO_UNICODE[20461] := 16#7DC8;
   // GBK_TO_UNICODE[20462] := 16#BE6E;
   // GBK_TO_UNICODE[20463] := 16#7DC9;
   // GBK_TO_UNICODE[20464] := 16#BE6F;
   // GBK_TO_UNICODE[20465] := 16#7DCA;
   // GBK_TO_UNICODE[20466] := 16#BE70;
   // GBK_TO_UNICODE[20467] := 16#7DCB;
   // GBK_TO_UNICODE[20468] := 16#BE71;
   // GBK_TO_UNICODE[20469] := 16#7DCC;
   // GBK_TO_UNICODE[20470] := 16#BE72;
   // GBK_TO_UNICODE[20471] := 16#7DCD;
   // GBK_TO_UNICODE[20472] := 16#BE73;
   // GBK_TO_UNICODE[20473] := 16#7DCE;
   // GBK_TO_UNICODE[20474] := 16#BE74;
   // GBK_TO_UNICODE[20475] := 16#7DCF;
   // GBK_TO_UNICODE[20476] := 16#BE75;
   // GBK_TO_UNICODE[20477] := 16#7DD0;
   // GBK_TO_UNICODE[20478] := 16#BE76;
   // GBK_TO_UNICODE[20479] := 16#7DD1;
   // GBK_TO_UNICODE[20480] := 16#BE77;
   // GBK_TO_UNICODE[20481] := 16#7DD2;
   // GBK_TO_UNICODE[20482] := 16#BE78;
   // GBK_TO_UNICODE[20483] := 16#7DD3;
   // GBK_TO_UNICODE[20484] := 16#BE79;
   // GBK_TO_UNICODE[20485] := 16#7DD4;
   // GBK_TO_UNICODE[20486] := 16#BE7A;
   // GBK_TO_UNICODE[20487] := 16#7DD5;
   // GBK_TO_UNICODE[20488] := 16#BE7B;
   // GBK_TO_UNICODE[20489] := 16#7DD6;
   // GBK_TO_UNICODE[20490] := 16#BE7C;
   // GBK_TO_UNICODE[20491] := 16#7DD7;
   // GBK_TO_UNICODE[20492] := 16#BE7D;
   // GBK_TO_UNICODE[20493] := 16#7DD8;
   // GBK_TO_UNICODE[20494] := 16#BE7E;
   // GBK_TO_UNICODE[20495] := 16#7DD9;
   // GBK_TO_UNICODE[20496] := 16#BE80;
   // GBK_TO_UNICODE[20497] := 16#7DDA;
   // GBK_TO_UNICODE[20498] := 16#BE81;
   // GBK_TO_UNICODE[20499] := 16#7DDB;
   // GBK_TO_UNICODE[20500] := 16#BE82;
   // GBK_TO_UNICODE[20501] := 16#7DDC;
   // GBK_TO_UNICODE[20502] := 16#BE83;
   // GBK_TO_UNICODE[20503] := 16#7DDD;
   // GBK_TO_UNICODE[20504] := 16#BE84;
   // GBK_TO_UNICODE[20505] := 16#7DDE;
   // GBK_TO_UNICODE[20506] := 16#BE85;
   // GBK_TO_UNICODE[20507] := 16#7DDF;
   // GBK_TO_UNICODE[20508] := 16#BE86;
   // GBK_TO_UNICODE[20509] := 16#7DE0;
   // GBK_TO_UNICODE[20510] := 16#BE87;
   // GBK_TO_UNICODE[20511] := 16#7DE1;
   // GBK_TO_UNICODE[20512] := 16#BE88;
   // GBK_TO_UNICODE[20513] := 16#7DE2;
   // GBK_TO_UNICODE[20514] := 16#BE89;
   // GBK_TO_UNICODE[20515] := 16#7DE3;
   // GBK_TO_UNICODE[20516] := 16#BE8A;
   // GBK_TO_UNICODE[20517] := 16#7DE4;
   // GBK_TO_UNICODE[20518] := 16#BE8B;
   // GBK_TO_UNICODE[20519] := 16#7DE5;
   // GBK_TO_UNICODE[20520] := 16#BE8C;
   // GBK_TO_UNICODE[20521] := 16#7DE6;
   // GBK_TO_UNICODE[20522] := 16#BE8D;
   // GBK_TO_UNICODE[20523] := 16#7DE7;
   // GBK_TO_UNICODE[20524] := 16#BE8E;
   // GBK_TO_UNICODE[20525] := 16#7DE8;
   // GBK_TO_UNICODE[20526] := 16#BE8F;
   // GBK_TO_UNICODE[20527] := 16#7DE9;
   // GBK_TO_UNICODE[20528] := 16#BE90;
   // GBK_TO_UNICODE[20529] := 16#7DEA;
   // GBK_TO_UNICODE[20530] := 16#BE91;
   // GBK_TO_UNICODE[20531] := 16#7DEB;
   // GBK_TO_UNICODE[20532] := 16#BE92;
   // GBK_TO_UNICODE[20533] := 16#7DEC;
   // GBK_TO_UNICODE[20534] := 16#BE93;
   // GBK_TO_UNICODE[20535] := 16#7DED;
   // GBK_TO_UNICODE[20536] := 16#BE94;
   // GBK_TO_UNICODE[20537] := 16#7DEE;
   // GBK_TO_UNICODE[20538] := 16#BE95;
   // GBK_TO_UNICODE[20539] := 16#7DEF;
   // GBK_TO_UNICODE[20540] := 16#BE96;
   // GBK_TO_UNICODE[20541] := 16#7DF0;
   // GBK_TO_UNICODE[20542] := 16#BE97;
   // GBK_TO_UNICODE[20543] := 16#7DF1;
   // GBK_TO_UNICODE[20544] := 16#BE98;
   // GBK_TO_UNICODE[20545] := 16#7DF2;
   // GBK_TO_UNICODE[20546] := 16#BE99;
   // GBK_TO_UNICODE[20547] := 16#7DF3;
   // GBK_TO_UNICODE[20548] := 16#BE9A;
   // GBK_TO_UNICODE[20549] := 16#7DF4;
   // GBK_TO_UNICODE[20550] := 16#BE9B;
   // GBK_TO_UNICODE[20551] := 16#7DF5;
   // GBK_TO_UNICODE[20552] := 16#BE9C;
   // GBK_TO_UNICODE[20553] := 16#7DF6;
   // GBK_TO_UNICODE[20554] := 16#BE9D;
   // GBK_TO_UNICODE[20555] := 16#7DF7;
   // GBK_TO_UNICODE[20556] := 16#BE9E;
   // GBK_TO_UNICODE[20557] := 16#7DF8;
   // GBK_TO_UNICODE[20558] := 16#BE9F;
   // GBK_TO_UNICODE[20559] := 16#7DF9;
   // GBK_TO_UNICODE[20560] := 16#BEA0;
   // GBK_TO_UNICODE[20561] := 16#7DFA;
   // GBK_TO_UNICODE[20562] := 16#BEA1;
   // GBK_TO_UNICODE[20563] := 16#5C3D;
   // GBK_TO_UNICODE[20564] := 16#BEA2;
   // GBK_TO_UNICODE[20565] := 16#52B2;
   // GBK_TO_UNICODE[20566] := 16#BEA3;
   // GBK_TO_UNICODE[20567] := 16#8346;
   // GBK_TO_UNICODE[20568] := 16#BEA4;
   // GBK_TO_UNICODE[20569] := 16#5162;
   // GBK_TO_UNICODE[20570] := 16#BEA5;
   // GBK_TO_UNICODE[20571] := 16#830E;
   // GBK_TO_UNICODE[20572] := 16#BEA6;
   // GBK_TO_UNICODE[20573] := 16#775B;
   // GBK_TO_UNICODE[20574] := 16#BEA7;
   // GBK_TO_UNICODE[20575] := 16#6676;
   // GBK_TO_UNICODE[20576] := 16#BEA8;
   // GBK_TO_UNICODE[20577] := 16#9CB8;
   // GBK_TO_UNICODE[20578] := 16#BEA9;
   // GBK_TO_UNICODE[20579] := 16#4EAC;
   // GBK_TO_UNICODE[20580] := 16#BEAA;
   // GBK_TO_UNICODE[20581] := 16#60CA;
   // GBK_TO_UNICODE[20582] := 16#BEAB;
   // GBK_TO_UNICODE[20583] := 16#7CBE;
   // GBK_TO_UNICODE[20584] := 16#BEAC;
   // GBK_TO_UNICODE[20585] := 16#7CB3;
   // GBK_TO_UNICODE[20586] := 16#BEAD;
   // GBK_TO_UNICODE[20587] := 16#7ECF;
   // GBK_TO_UNICODE[20588] := 16#BEAE;
   // GBK_TO_UNICODE[20589] := 16#4E95;
   // GBK_TO_UNICODE[20590] := 16#BEAF;
   // GBK_TO_UNICODE[20591] := 16#8B66;
   // GBK_TO_UNICODE[20592] := 16#BEB0;
   // GBK_TO_UNICODE[20593] := 16#666F;
   // GBK_TO_UNICODE[20594] := 16#BEB1;
   // GBK_TO_UNICODE[20595] := 16#9888;
   // GBK_TO_UNICODE[20596] := 16#BEB2;
   // GBK_TO_UNICODE[20597] := 16#9759;
   // GBK_TO_UNICODE[20598] := 16#BEB3;
   // GBK_TO_UNICODE[20599] := 16#5883;
   // GBK_TO_UNICODE[20600] := 16#BEB4;
   // GBK_TO_UNICODE[20601] := 16#656C;
   // GBK_TO_UNICODE[20602] := 16#BEB5;
   // GBK_TO_UNICODE[20603] := 16#955C;
   // GBK_TO_UNICODE[20604] := 16#BEB6;
   // GBK_TO_UNICODE[20605] := 16#5F84;
   // GBK_TO_UNICODE[20606] := 16#BEB7;
   // GBK_TO_UNICODE[20607] := 16#75C9;
   // GBK_TO_UNICODE[20608] := 16#BEB8;
   // GBK_TO_UNICODE[20609] := 16#9756;
   // GBK_TO_UNICODE[20610] := 16#BEB9;
   // GBK_TO_UNICODE[20611] := 16#7ADF;
   // GBK_TO_UNICODE[20612] := 16#BEBA;
   // GBK_TO_UNICODE[20613] := 16#7ADE;
   // GBK_TO_UNICODE[20614] := 16#BEBB;
   // GBK_TO_UNICODE[20615] := 16#51C0;
   // GBK_TO_UNICODE[20616] := 16#BEBC;
   // GBK_TO_UNICODE[20617] := 16#70AF;
   // GBK_TO_UNICODE[20618] := 16#BEBD;
   // GBK_TO_UNICODE[20619] := 16#7A98;
   // GBK_TO_UNICODE[20620] := 16#BEBE;
   // GBK_TO_UNICODE[20621] := 16#63EA;
   // GBK_TO_UNICODE[20622] := 16#BEBF;
   // GBK_TO_UNICODE[20623] := 16#7A76;
   // GBK_TO_UNICODE[20624] := 16#BEC0;
   // GBK_TO_UNICODE[20625] := 16#7EA0;
   // GBK_TO_UNICODE[20626] := 16#BEC1;
   // GBK_TO_UNICODE[20627] := 16#7396;
   // GBK_TO_UNICODE[20628] := 16#BEC2;
   // GBK_TO_UNICODE[20629] := 16#97ED;
   // GBK_TO_UNICODE[20630] := 16#BEC3;
   // GBK_TO_UNICODE[20631] := 16#4E45;
   // GBK_TO_UNICODE[20632] := 16#BEC4;
   // GBK_TO_UNICODE[20633] := 16#7078;
   // GBK_TO_UNICODE[20634] := 16#BEC5;
   // GBK_TO_UNICODE[20635] := 16#4E5D;
   // GBK_TO_UNICODE[20636] := 16#BEC6;
   // GBK_TO_UNICODE[20637] := 16#9152;
   // GBK_TO_UNICODE[20638] := 16#BEC7;
   // GBK_TO_UNICODE[20639] := 16#53A9;
   // GBK_TO_UNICODE[20640] := 16#BEC8;
   // GBK_TO_UNICODE[20641] := 16#6551;
   // GBK_TO_UNICODE[20642] := 16#BEC9;
   // GBK_TO_UNICODE[20643] := 16#65E7;
   // GBK_TO_UNICODE[20644] := 16#BECA;
   // GBK_TO_UNICODE[20645] := 16#81FC;
   // GBK_TO_UNICODE[20646] := 16#BECB;
   // GBK_TO_UNICODE[20647] := 16#8205;
   // GBK_TO_UNICODE[20648] := 16#BECC;
   // GBK_TO_UNICODE[20649] := 16#548E;
   // GBK_TO_UNICODE[20650] := 16#BECD;
   // GBK_TO_UNICODE[20651] := 16#5C31;
   // GBK_TO_UNICODE[20652] := 16#BECE;
   // GBK_TO_UNICODE[20653] := 16#759A;
   // GBK_TO_UNICODE[20654] := 16#BECF;
   // GBK_TO_UNICODE[20655] := 16#97A0;
   // GBK_TO_UNICODE[20656] := 16#BED0;
   // GBK_TO_UNICODE[20657] := 16#62D8;
   // GBK_TO_UNICODE[20658] := 16#BED1;
   // GBK_TO_UNICODE[20659] := 16#72D9;
   // GBK_TO_UNICODE[20660] := 16#BED2;
   // GBK_TO_UNICODE[20661] := 16#75BD;
   // GBK_TO_UNICODE[20662] := 16#BED3;
   // GBK_TO_UNICODE[20663] := 16#5C45;
   // GBK_TO_UNICODE[20664] := 16#BED4;
   // GBK_TO_UNICODE[20665] := 16#9A79;
   // GBK_TO_UNICODE[20666] := 16#BED5;
   // GBK_TO_UNICODE[20667] := 16#83CA;
   // GBK_TO_UNICODE[20668] := 16#BED6;
   // GBK_TO_UNICODE[20669] := 16#5C40;
   // GBK_TO_UNICODE[20670] := 16#BED7;
   // GBK_TO_UNICODE[20671] := 16#5480;
   // GBK_TO_UNICODE[20672] := 16#BED8;
   // GBK_TO_UNICODE[20673] := 16#77E9;
   // GBK_TO_UNICODE[20674] := 16#BED9;
   // GBK_TO_UNICODE[20675] := 16#4E3E;
   // GBK_TO_UNICODE[20676] := 16#BEDA;
   // GBK_TO_UNICODE[20677] := 16#6CAE;
   // GBK_TO_UNICODE[20678] := 16#BEDB;
   // GBK_TO_UNICODE[20679] := 16#805A;
   // GBK_TO_UNICODE[20680] := 16#BEDC;
   // GBK_TO_UNICODE[20681] := 16#62D2;
   // GBK_TO_UNICODE[20682] := 16#BEDD;
   // GBK_TO_UNICODE[20683] := 16#636E;
   // GBK_TO_UNICODE[20684] := 16#BEDE;
   // GBK_TO_UNICODE[20685] := 16#5DE8;
   // GBK_TO_UNICODE[20686] := 16#BEDF;
   // GBK_TO_UNICODE[20687] := 16#5177;
   // GBK_TO_UNICODE[20688] := 16#BEE0;
   // GBK_TO_UNICODE[20689] := 16#8DDD;
   // GBK_TO_UNICODE[20690] := 16#BEE1;
   // GBK_TO_UNICODE[20691] := 16#8E1E;
   // GBK_TO_UNICODE[20692] := 16#BEE2;
   // GBK_TO_UNICODE[20693] := 16#952F;
   // GBK_TO_UNICODE[20694] := 16#BEE3;
   // GBK_TO_UNICODE[20695] := 16#4FF1;
   // GBK_TO_UNICODE[20696] := 16#BEE4;
   // GBK_TO_UNICODE[20697] := 16#53E5;
   // GBK_TO_UNICODE[20698] := 16#BEE5;
   // GBK_TO_UNICODE[20699] := 16#60E7;
   // GBK_TO_UNICODE[20700] := 16#BEE6;
   // GBK_TO_UNICODE[20701] := 16#70AC;
   // GBK_TO_UNICODE[20702] := 16#BEE7;
   // GBK_TO_UNICODE[20703] := 16#5267;
   // GBK_TO_UNICODE[20704] := 16#BEE8;
   // GBK_TO_UNICODE[20705] := 16#6350;
   // GBK_TO_UNICODE[20706] := 16#BEE9;
   // GBK_TO_UNICODE[20707] := 16#9E43;
   // GBK_TO_UNICODE[20708] := 16#BEEA;
   // GBK_TO_UNICODE[20709] := 16#5A1F;
   // GBK_TO_UNICODE[20710] := 16#BEEB;
   // GBK_TO_UNICODE[20711] := 16#5026;
   // GBK_TO_UNICODE[20712] := 16#BEEC;
   // GBK_TO_UNICODE[20713] := 16#7737;
   // GBK_TO_UNICODE[20714] := 16#BEED;
   // GBK_TO_UNICODE[20715] := 16#5377;
   // GBK_TO_UNICODE[20716] := 16#BEEE;
   // GBK_TO_UNICODE[20717] := 16#7EE2;
   // GBK_TO_UNICODE[20718] := 16#BEEF;
   // GBK_TO_UNICODE[20719] := 16#6485;
   // GBK_TO_UNICODE[20720] := 16#BEF0;
   // GBK_TO_UNICODE[20721] := 16#652B;
   // GBK_TO_UNICODE[20722] := 16#BEF1;
   // GBK_TO_UNICODE[20723] := 16#6289;
   // GBK_TO_UNICODE[20724] := 16#BEF2;
   // GBK_TO_UNICODE[20725] := 16#6398;
   // GBK_TO_UNICODE[20726] := 16#BEF3;
   // GBK_TO_UNICODE[20727] := 16#5014;
   // GBK_TO_UNICODE[20728] := 16#BEF4;
   // GBK_TO_UNICODE[20729] := 16#7235;
   // GBK_TO_UNICODE[20730] := 16#BEF5;
   // GBK_TO_UNICODE[20731] := 16#89C9;
   // GBK_TO_UNICODE[20732] := 16#BEF6;
   // GBK_TO_UNICODE[20733] := 16#51B3;
   // GBK_TO_UNICODE[20734] := 16#BEF7;
   // GBK_TO_UNICODE[20735] := 16#8BC0;
   // GBK_TO_UNICODE[20736] := 16#BEF8;
   // GBK_TO_UNICODE[20737] := 16#7EDD;
   // GBK_TO_UNICODE[20738] := 16#BEF9;
   // GBK_TO_UNICODE[20739] := 16#5747;
   // GBK_TO_UNICODE[20740] := 16#BEFA;
   // GBK_TO_UNICODE[20741] := 16#83CC;
   // GBK_TO_UNICODE[20742] := 16#BEFB;
   // GBK_TO_UNICODE[20743] := 16#94A7;
   // GBK_TO_UNICODE[20744] := 16#BEFC;
   // GBK_TO_UNICODE[20745] := 16#519B;
   // GBK_TO_UNICODE[20746] := 16#BEFD;
   // GBK_TO_UNICODE[20747] := 16#541B;
   // GBK_TO_UNICODE[20748] := 16#BEFE;
   // GBK_TO_UNICODE[20749] := 16#5CFB;
   // GBK_TO_UNICODE[20750] := 16#BF40;
   // GBK_TO_UNICODE[20751] := 16#7DFB;
   // GBK_TO_UNICODE[20752] := 16#BF41;
   // GBK_TO_UNICODE[20753] := 16#7DFC;
   // GBK_TO_UNICODE[20754] := 16#BF42;
   // GBK_TO_UNICODE[20755] := 16#7DFD;
   // GBK_TO_UNICODE[20756] := 16#BF43;
   // GBK_TO_UNICODE[20757] := 16#7DFE;
   // GBK_TO_UNICODE[20758] := 16#BF44;
   // GBK_TO_UNICODE[20759] := 16#7DFF;
   // GBK_TO_UNICODE[20760] := 16#BF45;
   // GBK_TO_UNICODE[20761] := 16#7E00;
   // GBK_TO_UNICODE[20762] := 16#BF46;
   // GBK_TO_UNICODE[20763] := 16#7E01;
   // GBK_TO_UNICODE[20764] := 16#BF47;
   // GBK_TO_UNICODE[20765] := 16#7E02;
   // GBK_TO_UNICODE[20766] := 16#BF48;
   // GBK_TO_UNICODE[20767] := 16#7E03;
   // GBK_TO_UNICODE[20768] := 16#BF49;
   // GBK_TO_UNICODE[20769] := 16#7E04;
   // GBK_TO_UNICODE[20770] := 16#BF4A;
   // GBK_TO_UNICODE[20771] := 16#7E05;
   // GBK_TO_UNICODE[20772] := 16#BF4B;
   // GBK_TO_UNICODE[20773] := 16#7E06;
   // GBK_TO_UNICODE[20774] := 16#BF4C;
   // GBK_TO_UNICODE[20775] := 16#7E07;
   // GBK_TO_UNICODE[20776] := 16#BF4D;
   // GBK_TO_UNICODE[20777] := 16#7E08;
   // GBK_TO_UNICODE[20778] := 16#BF4E;
   // GBK_TO_UNICODE[20779] := 16#7E09;
   // GBK_TO_UNICODE[20780] := 16#BF4F;
   // GBK_TO_UNICODE[20781] := 16#7E0A;
   // GBK_TO_UNICODE[20782] := 16#BF50;
   // GBK_TO_UNICODE[20783] := 16#7E0B;
   // GBK_TO_UNICODE[20784] := 16#BF51;
   // GBK_TO_UNICODE[20785] := 16#7E0C;
   // GBK_TO_UNICODE[20786] := 16#BF52;
   // GBK_TO_UNICODE[20787] := 16#7E0D;
   // GBK_TO_UNICODE[20788] := 16#BF53;
   // GBK_TO_UNICODE[20789] := 16#7E0E;
   // GBK_TO_UNICODE[20790] := 16#BF54;
   // GBK_TO_UNICODE[20791] := 16#7E0F;
   // GBK_TO_UNICODE[20792] := 16#BF55;
   // GBK_TO_UNICODE[20793] := 16#7E10;
   // GBK_TO_UNICODE[20794] := 16#BF56;
   // GBK_TO_UNICODE[20795] := 16#7E11;
   // GBK_TO_UNICODE[20796] := 16#BF57;
   // GBK_TO_UNICODE[20797] := 16#7E12;
   // GBK_TO_UNICODE[20798] := 16#BF58;
   // GBK_TO_UNICODE[20799] := 16#7E13;
   // GBK_TO_UNICODE[20800] := 16#BF59;
   // GBK_TO_UNICODE[20801] := 16#7E14;
   // GBK_TO_UNICODE[20802] := 16#BF5A;
   // GBK_TO_UNICODE[20803] := 16#7E15;
   // GBK_TO_UNICODE[20804] := 16#BF5B;
   // GBK_TO_UNICODE[20805] := 16#7E16;
   // GBK_TO_UNICODE[20806] := 16#BF5C;
   // GBK_TO_UNICODE[20807] := 16#7E17;
   // GBK_TO_UNICODE[20808] := 16#BF5D;
   // GBK_TO_UNICODE[20809] := 16#7E18;
   // GBK_TO_UNICODE[20810] := 16#BF5E;
   // GBK_TO_UNICODE[20811] := 16#7E19;
   // GBK_TO_UNICODE[20812] := 16#BF5F;
   // GBK_TO_UNICODE[20813] := 16#7E1A;
   // GBK_TO_UNICODE[20814] := 16#BF60;
   // GBK_TO_UNICODE[20815] := 16#7E1B;
   // GBK_TO_UNICODE[20816] := 16#BF61;
   // GBK_TO_UNICODE[20817] := 16#7E1C;
   // GBK_TO_UNICODE[20818] := 16#BF62;
   // GBK_TO_UNICODE[20819] := 16#7E1D;
   // GBK_TO_UNICODE[20820] := 16#BF63;
   // GBK_TO_UNICODE[20821] := 16#7E1E;
   // GBK_TO_UNICODE[20822] := 16#BF64;
   // GBK_TO_UNICODE[20823] := 16#7E1F;
   // GBK_TO_UNICODE[20824] := 16#BF65;
   // GBK_TO_UNICODE[20825] := 16#7E20;
   // GBK_TO_UNICODE[20826] := 16#BF66;
   // GBK_TO_UNICODE[20827] := 16#7E21;
   // GBK_TO_UNICODE[20828] := 16#BF67;
   // GBK_TO_UNICODE[20829] := 16#7E22;
   // GBK_TO_UNICODE[20830] := 16#BF68;
   // GBK_TO_UNICODE[20831] := 16#7E23;
   // GBK_TO_UNICODE[20832] := 16#BF69;
   // GBK_TO_UNICODE[20833] := 16#7E24;
   // GBK_TO_UNICODE[20834] := 16#BF6A;
   // GBK_TO_UNICODE[20835] := 16#7E25;
   // GBK_TO_UNICODE[20836] := 16#BF6B;
   // GBK_TO_UNICODE[20837] := 16#7E26;
   // GBK_TO_UNICODE[20838] := 16#BF6C;
   // GBK_TO_UNICODE[20839] := 16#7E27;
   // GBK_TO_UNICODE[20840] := 16#BF6D;
   // GBK_TO_UNICODE[20841] := 16#7E28;
   // GBK_TO_UNICODE[20842] := 16#BF6E;
   // GBK_TO_UNICODE[20843] := 16#7E29;
   // GBK_TO_UNICODE[20844] := 16#BF6F;
   // GBK_TO_UNICODE[20845] := 16#7E2A;
   // GBK_TO_UNICODE[20846] := 16#BF70;
   // GBK_TO_UNICODE[20847] := 16#7E2B;
   // GBK_TO_UNICODE[20848] := 16#BF71;
   // GBK_TO_UNICODE[20849] := 16#7E2C;
   // GBK_TO_UNICODE[20850] := 16#BF72;
   // GBK_TO_UNICODE[20851] := 16#7E2D;
   // GBK_TO_UNICODE[20852] := 16#BF73;
   // GBK_TO_UNICODE[20853] := 16#7E2E;
   // GBK_TO_UNICODE[20854] := 16#BF74;
   // GBK_TO_UNICODE[20855] := 16#7E2F;
   // GBK_TO_UNICODE[20856] := 16#BF75;
   // GBK_TO_UNICODE[20857] := 16#7E30;
   // GBK_TO_UNICODE[20858] := 16#BF76;
   // GBK_TO_UNICODE[20859] := 16#7E31;
   // GBK_TO_UNICODE[20860] := 16#BF77;
   // GBK_TO_UNICODE[20861] := 16#7E32;
   // GBK_TO_UNICODE[20862] := 16#BF78;
   // GBK_TO_UNICODE[20863] := 16#7E33;
   // GBK_TO_UNICODE[20864] := 16#BF79;
   // GBK_TO_UNICODE[20865] := 16#7E34;
   // GBK_TO_UNICODE[20866] := 16#BF7A;
   // GBK_TO_UNICODE[20867] := 16#7E35;
   // GBK_TO_UNICODE[20868] := 16#BF7B;
   // GBK_TO_UNICODE[20869] := 16#7E36;
   // GBK_TO_UNICODE[20870] := 16#BF7C;
   // GBK_TO_UNICODE[20871] := 16#7E37;
   // GBK_TO_UNICODE[20872] := 16#BF7D;
   // GBK_TO_UNICODE[20873] := 16#7E38;
   // GBK_TO_UNICODE[20874] := 16#BF7E;
   // GBK_TO_UNICODE[20875] := 16#7E39;
   // GBK_TO_UNICODE[20876] := 16#BF80;
   // GBK_TO_UNICODE[20877] := 16#7E3A;
   // GBK_TO_UNICODE[20878] := 16#BF81;
   // GBK_TO_UNICODE[20879] := 16#7E3C;
   // GBK_TO_UNICODE[20880] := 16#BF82;
   // GBK_TO_UNICODE[20881] := 16#7E3D;
   // GBK_TO_UNICODE[20882] := 16#BF83;
   // GBK_TO_UNICODE[20883] := 16#7E3E;
   // GBK_TO_UNICODE[20884] := 16#BF84;
   // GBK_TO_UNICODE[20885] := 16#7E3F;
   // GBK_TO_UNICODE[20886] := 16#BF85;
   // GBK_TO_UNICODE[20887] := 16#7E40;
   // GBK_TO_UNICODE[20888] := 16#BF86;
   // GBK_TO_UNICODE[20889] := 16#7E42;
   // GBK_TO_UNICODE[20890] := 16#BF87;
   // GBK_TO_UNICODE[20891] := 16#7E43;
   // GBK_TO_UNICODE[20892] := 16#BF88;
   // GBK_TO_UNICODE[20893] := 16#7E44;
   // GBK_TO_UNICODE[20894] := 16#BF89;
   // GBK_TO_UNICODE[20895] := 16#7E45;
   // GBK_TO_UNICODE[20896] := 16#BF8A;
   // GBK_TO_UNICODE[20897] := 16#7E46;
   // GBK_TO_UNICODE[20898] := 16#BF8B;
   // GBK_TO_UNICODE[20899] := 16#7E48;
   // GBK_TO_UNICODE[20900] := 16#BF8C;
   // GBK_TO_UNICODE[20901] := 16#7E49;
   // GBK_TO_UNICODE[20902] := 16#BF8D;
   // GBK_TO_UNICODE[20903] := 16#7E4A;
   // GBK_TO_UNICODE[20904] := 16#BF8E;
   // GBK_TO_UNICODE[20905] := 16#7E4B;
   // GBK_TO_UNICODE[20906] := 16#BF8F;
   // GBK_TO_UNICODE[20907] := 16#7E4C;
   // GBK_TO_UNICODE[20908] := 16#BF90;
   // GBK_TO_UNICODE[20909] := 16#7E4D;
   // GBK_TO_UNICODE[20910] := 16#BF91;
   // GBK_TO_UNICODE[20911] := 16#7E4E;
   // GBK_TO_UNICODE[20912] := 16#BF92;
   // GBK_TO_UNICODE[20913] := 16#7E4F;
   // GBK_TO_UNICODE[20914] := 16#BF93;
   // GBK_TO_UNICODE[20915] := 16#7E50;
   // GBK_TO_UNICODE[20916] := 16#BF94;
   // GBK_TO_UNICODE[20917] := 16#7E51;
   // GBK_TO_UNICODE[20918] := 16#BF95;
   // GBK_TO_UNICODE[20919] := 16#7E52;
   // GBK_TO_UNICODE[20920] := 16#BF96;
   // GBK_TO_UNICODE[20921] := 16#7E53;
   // GBK_TO_UNICODE[20922] := 16#BF97;
   // GBK_TO_UNICODE[20923] := 16#7E54;
   // GBK_TO_UNICODE[20924] := 16#BF98;
   // GBK_TO_UNICODE[20925] := 16#7E55;
   // GBK_TO_UNICODE[20926] := 16#BF99;
   // GBK_TO_UNICODE[20927] := 16#7E56;
   // GBK_TO_UNICODE[20928] := 16#BF9A;
   // GBK_TO_UNICODE[20929] := 16#7E57;
   // GBK_TO_UNICODE[20930] := 16#BF9B;
   // GBK_TO_UNICODE[20931] := 16#7E58;
   // GBK_TO_UNICODE[20932] := 16#BF9C;
   // GBK_TO_UNICODE[20933] := 16#7E59;
   // GBK_TO_UNICODE[20934] := 16#BF9D;
   // GBK_TO_UNICODE[20935] := 16#7E5A;
   // GBK_TO_UNICODE[20936] := 16#BF9E;
   // GBK_TO_UNICODE[20937] := 16#7E5B;
   // GBK_TO_UNICODE[20938] := 16#BF9F;
   // GBK_TO_UNICODE[20939] := 16#7E5C;
   // GBK_TO_UNICODE[20940] := 16#BFA0;
   // GBK_TO_UNICODE[20941] := 16#7E5D;
   // GBK_TO_UNICODE[20942] := 16#BFA1;
   // GBK_TO_UNICODE[20943] := 16#4FCA;
   // GBK_TO_UNICODE[20944] := 16#BFA2;
   // GBK_TO_UNICODE[20945] := 16#7AE3;
   // GBK_TO_UNICODE[20946] := 16#BFA3;
   // GBK_TO_UNICODE[20947] := 16#6D5A;
   // GBK_TO_UNICODE[20948] := 16#BFA4;
   // GBK_TO_UNICODE[20949] := 16#90E1;
   // GBK_TO_UNICODE[20950] := 16#BFA5;
   // GBK_TO_UNICODE[20951] := 16#9A8F;
   // GBK_TO_UNICODE[20952] := 16#BFA6;
   // GBK_TO_UNICODE[20953] := 16#5580;
   // GBK_TO_UNICODE[20954] := 16#BFA7;
   // GBK_TO_UNICODE[20955] := 16#5496;
   // GBK_TO_UNICODE[20956] := 16#BFA8;
   // GBK_TO_UNICODE[20957] := 16#5361;
   // GBK_TO_UNICODE[20958] := 16#BFA9;
   // GBK_TO_UNICODE[20959] := 16#54AF;
   // GBK_TO_UNICODE[20960] := 16#BFAA;
   // GBK_TO_UNICODE[20961] := 16#5F00;
   // GBK_TO_UNICODE[20962] := 16#BFAB;
   // GBK_TO_UNICODE[20963] := 16#63E9;
   // GBK_TO_UNICODE[20964] := 16#BFAC;
   // GBK_TO_UNICODE[20965] := 16#6977;
   // GBK_TO_UNICODE[20966] := 16#BFAD;
   // GBK_TO_UNICODE[20967] := 16#51EF;
   // GBK_TO_UNICODE[20968] := 16#BFAE;
   // GBK_TO_UNICODE[20969] := 16#6168;
   // GBK_TO_UNICODE[20970] := 16#BFAF;
   // GBK_TO_UNICODE[20971] := 16#520A;
   // GBK_TO_UNICODE[20972] := 16#BFB0;
   // GBK_TO_UNICODE[20973] := 16#582A;
   // GBK_TO_UNICODE[20974] := 16#BFB1;
   // GBK_TO_UNICODE[20975] := 16#52D8;
   // GBK_TO_UNICODE[20976] := 16#BFB2;
   // GBK_TO_UNICODE[20977] := 16#574E;
   // GBK_TO_UNICODE[20978] := 16#BFB3;
   // GBK_TO_UNICODE[20979] := 16#780D;
   // GBK_TO_UNICODE[20980] := 16#BFB4;
   // GBK_TO_UNICODE[20981] := 16#770B;
   // GBK_TO_UNICODE[20982] := 16#BFB5;
   // GBK_TO_UNICODE[20983] := 16#5EB7;
   // GBK_TO_UNICODE[20984] := 16#BFB6;
   // GBK_TO_UNICODE[20985] := 16#6177;
   // GBK_TO_UNICODE[20986] := 16#BFB7;
   // GBK_TO_UNICODE[20987] := 16#7CE0;
   // GBK_TO_UNICODE[20988] := 16#BFB8;
   // GBK_TO_UNICODE[20989] := 16#625B;
   // GBK_TO_UNICODE[20990] := 16#BFB9;
   // GBK_TO_UNICODE[20991] := 16#6297;
   // GBK_TO_UNICODE[20992] := 16#BFBA;
   // GBK_TO_UNICODE[20993] := 16#4EA2;
   // GBK_TO_UNICODE[20994] := 16#BFBB;
   // GBK_TO_UNICODE[20995] := 16#7095;
   // GBK_TO_UNICODE[20996] := 16#BFBC;
   // GBK_TO_UNICODE[20997] := 16#8003;
   // GBK_TO_UNICODE[20998] := 16#BFBD;
   // GBK_TO_UNICODE[20999] := 16#62F7;
   // GBK_TO_UNICODE[21000] := 16#BFBE;
   // GBK_TO_UNICODE[21001] := 16#70E4;
   // GBK_TO_UNICODE[21002] := 16#BFBF;
   // GBK_TO_UNICODE[21003] := 16#9760;
   // GBK_TO_UNICODE[21004] := 16#BFC0;
   // GBK_TO_UNICODE[21005] := 16#5777;
   // GBK_TO_UNICODE[21006] := 16#BFC1;
   // GBK_TO_UNICODE[21007] := 16#82DB;
   // GBK_TO_UNICODE[21008] := 16#BFC2;
   // GBK_TO_UNICODE[21009] := 16#67EF;
   // GBK_TO_UNICODE[21010] := 16#BFC3;
   // GBK_TO_UNICODE[21011] := 16#68F5;
   // GBK_TO_UNICODE[21012] := 16#BFC4;
   // GBK_TO_UNICODE[21013] := 16#78D5;
   // GBK_TO_UNICODE[21014] := 16#BFC5;
   // GBK_TO_UNICODE[21015] := 16#9897;
   // GBK_TO_UNICODE[21016] := 16#BFC6;
   // GBK_TO_UNICODE[21017] := 16#79D1;
   // GBK_TO_UNICODE[21018] := 16#BFC7;
   // GBK_TO_UNICODE[21019] := 16#58F3;
   // GBK_TO_UNICODE[21020] := 16#BFC8;
   // GBK_TO_UNICODE[21021] := 16#54B3;
   // GBK_TO_UNICODE[21022] := 16#BFC9;
   // GBK_TO_UNICODE[21023] := 16#53EF;
   // GBK_TO_UNICODE[21024] := 16#BFCA;
   // GBK_TO_UNICODE[21025] := 16#6E34;
   // GBK_TO_UNICODE[21026] := 16#BFCB;
   // GBK_TO_UNICODE[21027] := 16#514B;
   // GBK_TO_UNICODE[21028] := 16#BFCC;
   // GBK_TO_UNICODE[21029] := 16#523B;
   // GBK_TO_UNICODE[21030] := 16#BFCD;
   // GBK_TO_UNICODE[21031] := 16#5BA2;
   // GBK_TO_UNICODE[21032] := 16#BFCE;
   // GBK_TO_UNICODE[21033] := 16#8BFE;
   // GBK_TO_UNICODE[21034] := 16#BFCF;
   // GBK_TO_UNICODE[21035] := 16#80AF;
   // GBK_TO_UNICODE[21036] := 16#BFD0;
   // GBK_TO_UNICODE[21037] := 16#5543;
   // GBK_TO_UNICODE[21038] := 16#BFD1;
   // GBK_TO_UNICODE[21039] := 16#57A6;
   // GBK_TO_UNICODE[21040] := 16#BFD2;
   // GBK_TO_UNICODE[21041] := 16#6073;
   // GBK_TO_UNICODE[21042] := 16#BFD3;
   // GBK_TO_UNICODE[21043] := 16#5751;
   // GBK_TO_UNICODE[21044] := 16#BFD4;
   // GBK_TO_UNICODE[21045] := 16#542D;
   // GBK_TO_UNICODE[21046] := 16#BFD5;
   // GBK_TO_UNICODE[21047] := 16#7A7A;
   // GBK_TO_UNICODE[21048] := 16#BFD6;
   // GBK_TO_UNICODE[21049] := 16#6050;
   // GBK_TO_UNICODE[21050] := 16#BFD7;
   // GBK_TO_UNICODE[21051] := 16#5B54;
   // GBK_TO_UNICODE[21052] := 16#BFD8;
   // GBK_TO_UNICODE[21053] := 16#63A7;
   // GBK_TO_UNICODE[21054] := 16#BFD9;
   // GBK_TO_UNICODE[21055] := 16#62A0;
   // GBK_TO_UNICODE[21056] := 16#BFDA;
   // GBK_TO_UNICODE[21057] := 16#53E3;
   // GBK_TO_UNICODE[21058] := 16#BFDB;
   // GBK_TO_UNICODE[21059] := 16#6263;
   // GBK_TO_UNICODE[21060] := 16#BFDC;
   // GBK_TO_UNICODE[21061] := 16#5BC7;
   // GBK_TO_UNICODE[21062] := 16#BFDD;
   // GBK_TO_UNICODE[21063] := 16#67AF;
   // GBK_TO_UNICODE[21064] := 16#BFDE;
   // GBK_TO_UNICODE[21065] := 16#54ED;
   // GBK_TO_UNICODE[21066] := 16#BFDF;
   // GBK_TO_UNICODE[21067] := 16#7A9F;
   // GBK_TO_UNICODE[21068] := 16#BFE0;
   // GBK_TO_UNICODE[21069] := 16#82E6;
   // GBK_TO_UNICODE[21070] := 16#BFE1;
   // GBK_TO_UNICODE[21071] := 16#9177;
   // GBK_TO_UNICODE[21072] := 16#BFE2;
   // GBK_TO_UNICODE[21073] := 16#5E93;
   // GBK_TO_UNICODE[21074] := 16#BFE3;
   // GBK_TO_UNICODE[21075] := 16#88E4;
   // GBK_TO_UNICODE[21076] := 16#BFE4;
   // GBK_TO_UNICODE[21077] := 16#5938;
   // GBK_TO_UNICODE[21078] := 16#BFE5;
   // GBK_TO_UNICODE[21079] := 16#57AE;
   // GBK_TO_UNICODE[21080] := 16#BFE6;
   // GBK_TO_UNICODE[21081] := 16#630E;
   // GBK_TO_UNICODE[21082] := 16#BFE7;
   // GBK_TO_UNICODE[21083] := 16#8DE8;
   // GBK_TO_UNICODE[21084] := 16#BFE8;
   // GBK_TO_UNICODE[21085] := 16#80EF;
   // GBK_TO_UNICODE[21086] := 16#BFE9;
   // GBK_TO_UNICODE[21087] := 16#5757;
   // GBK_TO_UNICODE[21088] := 16#BFEA;
   // GBK_TO_UNICODE[21089] := 16#7B77;
   // GBK_TO_UNICODE[21090] := 16#BFEB;
   // GBK_TO_UNICODE[21091] := 16#4FA9;
   // GBK_TO_UNICODE[21092] := 16#BFEC;
   // GBK_TO_UNICODE[21093] := 16#5FEB;
   // GBK_TO_UNICODE[21094] := 16#BFED;
   // GBK_TO_UNICODE[21095] := 16#5BBD;
   // GBK_TO_UNICODE[21096] := 16#BFEE;
   // GBK_TO_UNICODE[21097] := 16#6B3E;
   // GBK_TO_UNICODE[21098] := 16#BFEF;
   // GBK_TO_UNICODE[21099] := 16#5321;
   // GBK_TO_UNICODE[21100] := 16#BFF0;
   // GBK_TO_UNICODE[21101] := 16#7B50;
   // GBK_TO_UNICODE[21102] := 16#BFF1;
   // GBK_TO_UNICODE[21103] := 16#72C2;
   // GBK_TO_UNICODE[21104] := 16#BFF2;
   // GBK_TO_UNICODE[21105] := 16#6846;
   // GBK_TO_UNICODE[21106] := 16#BFF3;
   // GBK_TO_UNICODE[21107] := 16#77FF;
   // GBK_TO_UNICODE[21108] := 16#BFF4;
   // GBK_TO_UNICODE[21109] := 16#7736;
   // GBK_TO_UNICODE[21110] := 16#BFF5;
   // GBK_TO_UNICODE[21111] := 16#65F7;
   // GBK_TO_UNICODE[21112] := 16#BFF6;
   // GBK_TO_UNICODE[21113] := 16#51B5;
   // GBK_TO_UNICODE[21114] := 16#BFF7;
   // GBK_TO_UNICODE[21115] := 16#4E8F;
   // GBK_TO_UNICODE[21116] := 16#BFF8;
   // GBK_TO_UNICODE[21117] := 16#76D4;
   // GBK_TO_UNICODE[21118] := 16#BFF9;
   // GBK_TO_UNICODE[21119] := 16#5CBF;
   // GBK_TO_UNICODE[21120] := 16#BFFA;
   // GBK_TO_UNICODE[21121] := 16#7AA5;
   // GBK_TO_UNICODE[21122] := 16#BFFB;
   // GBK_TO_UNICODE[21123] := 16#8475;
   // GBK_TO_UNICODE[21124] := 16#BFFC;
   // GBK_TO_UNICODE[21125] := 16#594E;
   // GBK_TO_UNICODE[21126] := 16#BFFD;
   // GBK_TO_UNICODE[21127] := 16#9B41;
   // GBK_TO_UNICODE[21128] := 16#BFFE;
   // GBK_TO_UNICODE[21129] := 16#5080;
   // GBK_TO_UNICODE[21130] := 16#C040;
   // GBK_TO_UNICODE[21131] := 16#7E5E;
   // GBK_TO_UNICODE[21132] := 16#C041;
   // GBK_TO_UNICODE[21133] := 16#7E5F;
   // GBK_TO_UNICODE[21134] := 16#C042;
   // GBK_TO_UNICODE[21135] := 16#7E60;
   // GBK_TO_UNICODE[21136] := 16#C043;
   // GBK_TO_UNICODE[21137] := 16#7E61;
   // GBK_TO_UNICODE[21138] := 16#C044;
   // GBK_TO_UNICODE[21139] := 16#7E62;
   // GBK_TO_UNICODE[21140] := 16#C045;
   // GBK_TO_UNICODE[21141] := 16#7E63;
   // GBK_TO_UNICODE[21142] := 16#C046;
   // GBK_TO_UNICODE[21143] := 16#7E64;
   // GBK_TO_UNICODE[21144] := 16#C047;
   // GBK_TO_UNICODE[21145] := 16#7E65;
   // GBK_TO_UNICODE[21146] := 16#C048;
   // GBK_TO_UNICODE[21147] := 16#7E66;
   // GBK_TO_UNICODE[21148] := 16#C049;
   // GBK_TO_UNICODE[21149] := 16#7E67;
   // GBK_TO_UNICODE[21150] := 16#C04A;
   // GBK_TO_UNICODE[21151] := 16#7E68;
   // GBK_TO_UNICODE[21152] := 16#C04B;
   // GBK_TO_UNICODE[21153] := 16#7E69;
   // GBK_TO_UNICODE[21154] := 16#C04C;
   // GBK_TO_UNICODE[21155] := 16#7E6A;
   // GBK_TO_UNICODE[21156] := 16#C04D;
   // GBK_TO_UNICODE[21157] := 16#7E6B;
   // GBK_TO_UNICODE[21158] := 16#C04E;
   // GBK_TO_UNICODE[21159] := 16#7E6C;
   // GBK_TO_UNICODE[21160] := 16#C04F;
   // GBK_TO_UNICODE[21161] := 16#7E6D;
   // GBK_TO_UNICODE[21162] := 16#C050;
   // GBK_TO_UNICODE[21163] := 16#7E6E;
   // GBK_TO_UNICODE[21164] := 16#C051;
   // GBK_TO_UNICODE[21165] := 16#7E6F;
   // GBK_TO_UNICODE[21166] := 16#C052;
   // GBK_TO_UNICODE[21167] := 16#7E70;
   // GBK_TO_UNICODE[21168] := 16#C053;
   // GBK_TO_UNICODE[21169] := 16#7E71;
   // GBK_TO_UNICODE[21170] := 16#C054;
   // GBK_TO_UNICODE[21171] := 16#7E72;
   // GBK_TO_UNICODE[21172] := 16#C055;
   // GBK_TO_UNICODE[21173] := 16#7E73;
   // GBK_TO_UNICODE[21174] := 16#C056;
   // GBK_TO_UNICODE[21175] := 16#7E74;
   // GBK_TO_UNICODE[21176] := 16#C057;
   // GBK_TO_UNICODE[21177] := 16#7E75;
   // GBK_TO_UNICODE[21178] := 16#C058;
   // GBK_TO_UNICODE[21179] := 16#7E76;
   // GBK_TO_UNICODE[21180] := 16#C059;
   // GBK_TO_UNICODE[21181] := 16#7E77;
   // GBK_TO_UNICODE[21182] := 16#C05A;
   // GBK_TO_UNICODE[21183] := 16#7E78;
   // GBK_TO_UNICODE[21184] := 16#C05B;
   // GBK_TO_UNICODE[21185] := 16#7E79;
   // GBK_TO_UNICODE[21186] := 16#C05C;
   // GBK_TO_UNICODE[21187] := 16#7E7A;
   // GBK_TO_UNICODE[21188] := 16#C05D;
   // GBK_TO_UNICODE[21189] := 16#7E7B;
   // GBK_TO_UNICODE[21190] := 16#C05E;
   // GBK_TO_UNICODE[21191] := 16#7E7C;
   // GBK_TO_UNICODE[21192] := 16#C05F;
   // GBK_TO_UNICODE[21193] := 16#7E7D;
   // GBK_TO_UNICODE[21194] := 16#C060;
   // GBK_TO_UNICODE[21195] := 16#7E7E;
   // GBK_TO_UNICODE[21196] := 16#C061;
   // GBK_TO_UNICODE[21197] := 16#7E7F;
   // GBK_TO_UNICODE[21198] := 16#C062;
   // GBK_TO_UNICODE[21199] := 16#7E80;
   // GBK_TO_UNICODE[21200] := 16#C063;
   // GBK_TO_UNICODE[21201] := 16#7E81;
   // GBK_TO_UNICODE[21202] := 16#C064;
   // GBK_TO_UNICODE[21203] := 16#7E83;
   // GBK_TO_UNICODE[21204] := 16#C065;
   // GBK_TO_UNICODE[21205] := 16#7E84;
   // GBK_TO_UNICODE[21206] := 16#C066;
   // GBK_TO_UNICODE[21207] := 16#7E85;
   // GBK_TO_UNICODE[21208] := 16#C067;
   // GBK_TO_UNICODE[21209] := 16#7E86;
   // GBK_TO_UNICODE[21210] := 16#C068;
   // GBK_TO_UNICODE[21211] := 16#7E87;
   // GBK_TO_UNICODE[21212] := 16#C069;
   // GBK_TO_UNICODE[21213] := 16#7E88;
   // GBK_TO_UNICODE[21214] := 16#C06A;
   // GBK_TO_UNICODE[21215] := 16#7E89;
   // GBK_TO_UNICODE[21216] := 16#C06B;
   // GBK_TO_UNICODE[21217] := 16#7E8A;
   // GBK_TO_UNICODE[21218] := 16#C06C;
   // GBK_TO_UNICODE[21219] := 16#7E8B;
   // GBK_TO_UNICODE[21220] := 16#C06D;
   // GBK_TO_UNICODE[21221] := 16#7E8C;
   // GBK_TO_UNICODE[21222] := 16#C06E;
   // GBK_TO_UNICODE[21223] := 16#7E8D;
   // GBK_TO_UNICODE[21224] := 16#C06F;
   // GBK_TO_UNICODE[21225] := 16#7E8E;
   // GBK_TO_UNICODE[21226] := 16#C070;
   // GBK_TO_UNICODE[21227] := 16#7E8F;
   // GBK_TO_UNICODE[21228] := 16#C071;
   // GBK_TO_UNICODE[21229] := 16#7E90;
   // GBK_TO_UNICODE[21230] := 16#C072;
   // GBK_TO_UNICODE[21231] := 16#7E91;
   // GBK_TO_UNICODE[21232] := 16#C073;
   // GBK_TO_UNICODE[21233] := 16#7E92;
   // GBK_TO_UNICODE[21234] := 16#C074;
   // GBK_TO_UNICODE[21235] := 16#7E93;
   // GBK_TO_UNICODE[21236] := 16#C075;
   // GBK_TO_UNICODE[21237] := 16#7E94;
   // GBK_TO_UNICODE[21238] := 16#C076;
   // GBK_TO_UNICODE[21239] := 16#7E95;
   // GBK_TO_UNICODE[21240] := 16#C077;
   // GBK_TO_UNICODE[21241] := 16#7E96;
   // GBK_TO_UNICODE[21242] := 16#C078;
   // GBK_TO_UNICODE[21243] := 16#7E97;
   // GBK_TO_UNICODE[21244] := 16#C079;
   // GBK_TO_UNICODE[21245] := 16#7E98;
   // GBK_TO_UNICODE[21246] := 16#C07A;
   // GBK_TO_UNICODE[21247] := 16#7E99;
   // GBK_TO_UNICODE[21248] := 16#C07B;
   // GBK_TO_UNICODE[21249] := 16#7E9A;
   // GBK_TO_UNICODE[21250] := 16#C07C;
   // GBK_TO_UNICODE[21251] := 16#7E9C;
   // GBK_TO_UNICODE[21252] := 16#C07D;
   // GBK_TO_UNICODE[21253] := 16#7E9D;
   // GBK_TO_UNICODE[21254] := 16#C07E;
   // GBK_TO_UNICODE[21255] := 16#7E9E;
   // GBK_TO_UNICODE[21256] := 16#C080;
   // GBK_TO_UNICODE[21257] := 16#7EAE;
   // GBK_TO_UNICODE[21258] := 16#C081;
   // GBK_TO_UNICODE[21259] := 16#7EB4;
   // GBK_TO_UNICODE[21260] := 16#C082;
   // GBK_TO_UNICODE[21261] := 16#7EBB;
   // GBK_TO_UNICODE[21262] := 16#C083;
   // GBK_TO_UNICODE[21263] := 16#7EBC;
   // GBK_TO_UNICODE[21264] := 16#C084;
   // GBK_TO_UNICODE[21265] := 16#7ED6;
   // GBK_TO_UNICODE[21266] := 16#C085;
   // GBK_TO_UNICODE[21267] := 16#7EE4;
   // GBK_TO_UNICODE[21268] := 16#C086;
   // GBK_TO_UNICODE[21269] := 16#7EEC;
   // GBK_TO_UNICODE[21270] := 16#C087;
   // GBK_TO_UNICODE[21271] := 16#7EF9;
   // GBK_TO_UNICODE[21272] := 16#C088;
   // GBK_TO_UNICODE[21273] := 16#7F0A;
   // GBK_TO_UNICODE[21274] := 16#C089;
   // GBK_TO_UNICODE[21275] := 16#7F10;
   // GBK_TO_UNICODE[21276] := 16#C08A;
   // GBK_TO_UNICODE[21277] := 16#7F1E;
   // GBK_TO_UNICODE[21278] := 16#C08B;
   // GBK_TO_UNICODE[21279] := 16#7F37;
   // GBK_TO_UNICODE[21280] := 16#C08C;
   // GBK_TO_UNICODE[21281] := 16#7F39;
   // GBK_TO_UNICODE[21282] := 16#C08D;
   // GBK_TO_UNICODE[21283] := 16#7F3B;
   // GBK_TO_UNICODE[21284] := 16#C08E;
   // GBK_TO_UNICODE[21285] := 16#7F3C;
   // GBK_TO_UNICODE[21286] := 16#C08F;
   // GBK_TO_UNICODE[21287] := 16#7F3D;
   // GBK_TO_UNICODE[21288] := 16#C090;
   // GBK_TO_UNICODE[21289] := 16#7F3E;
   // GBK_TO_UNICODE[21290] := 16#C091;
   // GBK_TO_UNICODE[21291] := 16#7F3F;
   // GBK_TO_UNICODE[21292] := 16#C092;
   // GBK_TO_UNICODE[21293] := 16#7F40;
   // GBK_TO_UNICODE[21294] := 16#C093;
   // GBK_TO_UNICODE[21295] := 16#7F41;
   // GBK_TO_UNICODE[21296] := 16#C094;
   // GBK_TO_UNICODE[21297] := 16#7F43;
   // GBK_TO_UNICODE[21298] := 16#C095;
   // GBK_TO_UNICODE[21299] := 16#7F46;
   // GBK_TO_UNICODE[21300] := 16#C096;
   // GBK_TO_UNICODE[21301] := 16#7F47;
   // GBK_TO_UNICODE[21302] := 16#C097;
   // GBK_TO_UNICODE[21303] := 16#7F48;
   // GBK_TO_UNICODE[21304] := 16#C098;
   // GBK_TO_UNICODE[21305] := 16#7F49;
   // GBK_TO_UNICODE[21306] := 16#C099;
   // GBK_TO_UNICODE[21307] := 16#7F4A;
   // GBK_TO_UNICODE[21308] := 16#C09A;
   // GBK_TO_UNICODE[21309] := 16#7F4B;
   // GBK_TO_UNICODE[21310] := 16#C09B;
   // GBK_TO_UNICODE[21311] := 16#7F4C;
   // GBK_TO_UNICODE[21312] := 16#C09C;
   // GBK_TO_UNICODE[21313] := 16#7F4D;
   // GBK_TO_UNICODE[21314] := 16#C09D;
   // GBK_TO_UNICODE[21315] := 16#7F4E;
   // GBK_TO_UNICODE[21316] := 16#C09E;
   // GBK_TO_UNICODE[21317] := 16#7F4F;
   // GBK_TO_UNICODE[21318] := 16#C09F;
   // GBK_TO_UNICODE[21319] := 16#7F52;
   // GBK_TO_UNICODE[21320] := 16#C0A0;
   // GBK_TO_UNICODE[21321] := 16#7F53;
   // GBK_TO_UNICODE[21322] := 16#C0A1;
   // GBK_TO_UNICODE[21323] := 16#9988;
   // GBK_TO_UNICODE[21324] := 16#C0A2;
   // GBK_TO_UNICODE[21325] := 16#6127;
   // GBK_TO_UNICODE[21326] := 16#C0A3;
   // GBK_TO_UNICODE[21327] := 16#6E83;
   // GBK_TO_UNICODE[21328] := 16#C0A4;
   // GBK_TO_UNICODE[21329] := 16#5764;
   // GBK_TO_UNICODE[21330] := 16#C0A5;
   // GBK_TO_UNICODE[21331] := 16#6606;
   // GBK_TO_UNICODE[21332] := 16#C0A6;
   // GBK_TO_UNICODE[21333] := 16#6346;
   // GBK_TO_UNICODE[21334] := 16#C0A7;
   // GBK_TO_UNICODE[21335] := 16#56F0;
   // GBK_TO_UNICODE[21336] := 16#C0A8;
   // GBK_TO_UNICODE[21337] := 16#62EC;
   // GBK_TO_UNICODE[21338] := 16#C0A9;
   // GBK_TO_UNICODE[21339] := 16#6269;
   // GBK_TO_UNICODE[21340] := 16#C0AA;
   // GBK_TO_UNICODE[21341] := 16#5ED3;
   // GBK_TO_UNICODE[21342] := 16#C0AB;
   // GBK_TO_UNICODE[21343] := 16#9614;
   // GBK_TO_UNICODE[21344] := 16#C0AC;
   // GBK_TO_UNICODE[21345] := 16#5783;
   // GBK_TO_UNICODE[21346] := 16#C0AD;
   // GBK_TO_UNICODE[21347] := 16#62C9;
   // GBK_TO_UNICODE[21348] := 16#C0AE;
   // GBK_TO_UNICODE[21349] := 16#5587;
   // GBK_TO_UNICODE[21350] := 16#C0AF;
   // GBK_TO_UNICODE[21351] := 16#8721;
   // GBK_TO_UNICODE[21352] := 16#C0B0;
   // GBK_TO_UNICODE[21353] := 16#814A;
   // GBK_TO_UNICODE[21354] := 16#C0B1;
   // GBK_TO_UNICODE[21355] := 16#8FA3;
   // GBK_TO_UNICODE[21356] := 16#C0B2;
   // GBK_TO_UNICODE[21357] := 16#5566;
   // GBK_TO_UNICODE[21358] := 16#C0B3;
   // GBK_TO_UNICODE[21359] := 16#83B1;
   // GBK_TO_UNICODE[21360] := 16#C0B4;
   // GBK_TO_UNICODE[21361] := 16#6765;
   // GBK_TO_UNICODE[21362] := 16#C0B5;
   // GBK_TO_UNICODE[21363] := 16#8D56;
   // GBK_TO_UNICODE[21364] := 16#C0B6;
   // GBK_TO_UNICODE[21365] := 16#84DD;
   // GBK_TO_UNICODE[21366] := 16#C0B7;
   // GBK_TO_UNICODE[21367] := 16#5A6A;
   // GBK_TO_UNICODE[21368] := 16#C0B8;
   // GBK_TO_UNICODE[21369] := 16#680F;
   // GBK_TO_UNICODE[21370] := 16#C0B9;
   // GBK_TO_UNICODE[21371] := 16#62E6;
   // GBK_TO_UNICODE[21372] := 16#C0BA;
   // GBK_TO_UNICODE[21373] := 16#7BEE;
   // GBK_TO_UNICODE[21374] := 16#C0BB;
   // GBK_TO_UNICODE[21375] := 16#9611;
   // GBK_TO_UNICODE[21376] := 16#C0BC;
   // GBK_TO_UNICODE[21377] := 16#5170;
   // GBK_TO_UNICODE[21378] := 16#C0BD;
   // GBK_TO_UNICODE[21379] := 16#6F9C;
   // GBK_TO_UNICODE[21380] := 16#C0BE;
   // GBK_TO_UNICODE[21381] := 16#8C30;
   // GBK_TO_UNICODE[21382] := 16#C0BF;
   // GBK_TO_UNICODE[21383] := 16#63FD;
   // GBK_TO_UNICODE[21384] := 16#C0C0;
   // GBK_TO_UNICODE[21385] := 16#89C8;
   // GBK_TO_UNICODE[21386] := 16#C0C1;
   // GBK_TO_UNICODE[21387] := 16#61D2;
   // GBK_TO_UNICODE[21388] := 16#C0C2;
   // GBK_TO_UNICODE[21389] := 16#7F06;
   // GBK_TO_UNICODE[21390] := 16#C0C3;
   // GBK_TO_UNICODE[21391] := 16#70C2;
   // GBK_TO_UNICODE[21392] := 16#C0C4;
   // GBK_TO_UNICODE[21393] := 16#6EE5;
   // GBK_TO_UNICODE[21394] := 16#C0C5;
   // GBK_TO_UNICODE[21395] := 16#7405;
   // GBK_TO_UNICODE[21396] := 16#C0C6;
   // GBK_TO_UNICODE[21397] := 16#6994;
   // GBK_TO_UNICODE[21398] := 16#C0C7;
   // GBK_TO_UNICODE[21399] := 16#72FC;
   // GBK_TO_UNICODE[21400] := 16#C0C8;
   // GBK_TO_UNICODE[21401] := 16#5ECA;
   // GBK_TO_UNICODE[21402] := 16#C0C9;
   // GBK_TO_UNICODE[21403] := 16#90CE;
   // GBK_TO_UNICODE[21404] := 16#C0CA;
   // GBK_TO_UNICODE[21405] := 16#6717;
   // GBK_TO_UNICODE[21406] := 16#C0CB;
   // GBK_TO_UNICODE[21407] := 16#6D6A;
   // GBK_TO_UNICODE[21408] := 16#C0CC;
   // GBK_TO_UNICODE[21409] := 16#635E;
   // GBK_TO_UNICODE[21410] := 16#C0CD;
   // GBK_TO_UNICODE[21411] := 16#52B3;
   // GBK_TO_UNICODE[21412] := 16#C0CE;
   // GBK_TO_UNICODE[21413] := 16#7262;
   // GBK_TO_UNICODE[21414] := 16#C0CF;
   // GBK_TO_UNICODE[21415] := 16#8001;
   // GBK_TO_UNICODE[21416] := 16#C0D0;
   // GBK_TO_UNICODE[21417] := 16#4F6C;
   // GBK_TO_UNICODE[21418] := 16#C0D1;
   // GBK_TO_UNICODE[21419] := 16#59E5;
   // GBK_TO_UNICODE[21420] := 16#C0D2;
   // GBK_TO_UNICODE[21421] := 16#916A;
   // GBK_TO_UNICODE[21422] := 16#C0D3;
   // GBK_TO_UNICODE[21423] := 16#70D9;
   // GBK_TO_UNICODE[21424] := 16#C0D4;
   // GBK_TO_UNICODE[21425] := 16#6D9D;
   // GBK_TO_UNICODE[21426] := 16#C0D5;
   // GBK_TO_UNICODE[21427] := 16#52D2;
   // GBK_TO_UNICODE[21428] := 16#C0D6;
   // GBK_TO_UNICODE[21429] := 16#4E50;
   // GBK_TO_UNICODE[21430] := 16#C0D7;
   // GBK_TO_UNICODE[21431] := 16#96F7;
   // GBK_TO_UNICODE[21432] := 16#C0D8;
   // GBK_TO_UNICODE[21433] := 16#956D;
   // GBK_TO_UNICODE[21434] := 16#C0D9;
   // GBK_TO_UNICODE[21435] := 16#857E;
   // GBK_TO_UNICODE[21436] := 16#C0DA;
   // GBK_TO_UNICODE[21437] := 16#78CA;
   // GBK_TO_UNICODE[21438] := 16#C0DB;
   // GBK_TO_UNICODE[21439] := 16#7D2F;
   // GBK_TO_UNICODE[21440] := 16#C0DC;
   // GBK_TO_UNICODE[21441] := 16#5121;
   // GBK_TO_UNICODE[21442] := 16#C0DD;
   // GBK_TO_UNICODE[21443] := 16#5792;
   // GBK_TO_UNICODE[21444] := 16#C0DE;
   // GBK_TO_UNICODE[21445] := 16#64C2;
   // GBK_TO_UNICODE[21446] := 16#C0DF;
   // GBK_TO_UNICODE[21447] := 16#808B;
   // GBK_TO_UNICODE[21448] := 16#C0E0;
   // GBK_TO_UNICODE[21449] := 16#7C7B;
   // GBK_TO_UNICODE[21450] := 16#C0E1;
   // GBK_TO_UNICODE[21451] := 16#6CEA;
   // GBK_TO_UNICODE[21452] := 16#C0E2;
   // GBK_TO_UNICODE[21453] := 16#68F1;
   // GBK_TO_UNICODE[21454] := 16#C0E3;
   // GBK_TO_UNICODE[21455] := 16#695E;
   // GBK_TO_UNICODE[21456] := 16#C0E4;
   // GBK_TO_UNICODE[21457] := 16#51B7;
   // GBK_TO_UNICODE[21458] := 16#C0E5;
   // GBK_TO_UNICODE[21459] := 16#5398;
   // GBK_TO_UNICODE[21460] := 16#C0E6;
   // GBK_TO_UNICODE[21461] := 16#68A8;
   // GBK_TO_UNICODE[21462] := 16#C0E7;
   // GBK_TO_UNICODE[21463] := 16#7281;
   // GBK_TO_UNICODE[21464] := 16#C0E8;
   // GBK_TO_UNICODE[21465] := 16#9ECE;
   // GBK_TO_UNICODE[21466] := 16#C0E9;
   // GBK_TO_UNICODE[21467] := 16#7BF1;
   // GBK_TO_UNICODE[21468] := 16#C0EA;
   // GBK_TO_UNICODE[21469] := 16#72F8;
   // GBK_TO_UNICODE[21470] := 16#C0EB;
   // GBK_TO_UNICODE[21471] := 16#79BB;
   // GBK_TO_UNICODE[21472] := 16#C0EC;
   // GBK_TO_UNICODE[21473] := 16#6F13;
   // GBK_TO_UNICODE[21474] := 16#C0ED;
   // GBK_TO_UNICODE[21475] := 16#7406;
   // GBK_TO_UNICODE[21476] := 16#C0EE;
   // GBK_TO_UNICODE[21477] := 16#674E;
   // GBK_TO_UNICODE[21478] := 16#C0EF;
   // GBK_TO_UNICODE[21479] := 16#91CC;
   // GBK_TO_UNICODE[21480] := 16#C0F0;
   // GBK_TO_UNICODE[21481] := 16#9CA4;
   // GBK_TO_UNICODE[21482] := 16#C0F1;
   // GBK_TO_UNICODE[21483] := 16#793C;
   // GBK_TO_UNICODE[21484] := 16#C0F2;
   // GBK_TO_UNICODE[21485] := 16#8389;
   // GBK_TO_UNICODE[21486] := 16#C0F3;
   // GBK_TO_UNICODE[21487] := 16#8354;
   // GBK_TO_UNICODE[21488] := 16#C0F4;
   // GBK_TO_UNICODE[21489] := 16#540F;
   // GBK_TO_UNICODE[21490] := 16#C0F5;
   // GBK_TO_UNICODE[21491] := 16#6817;
   // GBK_TO_UNICODE[21492] := 16#C0F6;
   // GBK_TO_UNICODE[21493] := 16#4E3D;
   // GBK_TO_UNICODE[21494] := 16#C0F7;
   // GBK_TO_UNICODE[21495] := 16#5389;
   // GBK_TO_UNICODE[21496] := 16#C0F8;
   // GBK_TO_UNICODE[21497] := 16#52B1;
   // GBK_TO_UNICODE[21498] := 16#C0F9;
   // GBK_TO_UNICODE[21499] := 16#783E;
   // GBK_TO_UNICODE[21500] := 16#C0FA;
   // GBK_TO_UNICODE[21501] := 16#5386;
   // GBK_TO_UNICODE[21502] := 16#C0FB;
   // GBK_TO_UNICODE[21503] := 16#5229;
   // GBK_TO_UNICODE[21504] := 16#C0FC;
   // GBK_TO_UNICODE[21505] := 16#5088;
   // GBK_TO_UNICODE[21506] := 16#C0FD;
   // GBK_TO_UNICODE[21507] := 16#4F8B;
   // GBK_TO_UNICODE[21508] := 16#C0FE;
   // GBK_TO_UNICODE[21509] := 16#4FD0;
   // GBK_TO_UNICODE[21510] := 16#C140;
   // GBK_TO_UNICODE[21511] := 16#7F56;
   // GBK_TO_UNICODE[21512] := 16#C141;
   // GBK_TO_UNICODE[21513] := 16#7F59;
   // GBK_TO_UNICODE[21514] := 16#C142;
   // GBK_TO_UNICODE[21515] := 16#7F5B;
   // GBK_TO_UNICODE[21516] := 16#C143;
   // GBK_TO_UNICODE[21517] := 16#7F5C;
   // GBK_TO_UNICODE[21518] := 16#C144;
   // GBK_TO_UNICODE[21519] := 16#7F5D;
   // GBK_TO_UNICODE[21520] := 16#C145;
   // GBK_TO_UNICODE[21521] := 16#7F5E;
   // GBK_TO_UNICODE[21522] := 16#C146;
   // GBK_TO_UNICODE[21523] := 16#7F60;
   // GBK_TO_UNICODE[21524] := 16#C147;
   // GBK_TO_UNICODE[21525] := 16#7F63;
   // GBK_TO_UNICODE[21526] := 16#C148;
   // GBK_TO_UNICODE[21527] := 16#7F64;
   // GBK_TO_UNICODE[21528] := 16#C149;
   // GBK_TO_UNICODE[21529] := 16#7F65;
   // GBK_TO_UNICODE[21530] := 16#C14A;
   // GBK_TO_UNICODE[21531] := 16#7F66;
   // GBK_TO_UNICODE[21532] := 16#C14B;
   // GBK_TO_UNICODE[21533] := 16#7F67;
   // GBK_TO_UNICODE[21534] := 16#C14C;
   // GBK_TO_UNICODE[21535] := 16#7F6B;
   // GBK_TO_UNICODE[21536] := 16#C14D;
   // GBK_TO_UNICODE[21537] := 16#7F6C;
   // GBK_TO_UNICODE[21538] := 16#C14E;
   // GBK_TO_UNICODE[21539] := 16#7F6D;
   // GBK_TO_UNICODE[21540] := 16#C14F;
   // GBK_TO_UNICODE[21541] := 16#7F6F;
   // GBK_TO_UNICODE[21542] := 16#C150;
   // GBK_TO_UNICODE[21543] := 16#7F70;
   // GBK_TO_UNICODE[21544] := 16#C151;
   // GBK_TO_UNICODE[21545] := 16#7F73;
   // GBK_TO_UNICODE[21546] := 16#C152;
   // GBK_TO_UNICODE[21547] := 16#7F75;
   // GBK_TO_UNICODE[21548] := 16#C153;
   // GBK_TO_UNICODE[21549] := 16#7F76;
   // GBK_TO_UNICODE[21550] := 16#C154;
   // GBK_TO_UNICODE[21551] := 16#7F77;
   // GBK_TO_UNICODE[21552] := 16#C155;
   // GBK_TO_UNICODE[21553] := 16#7F78;
   // GBK_TO_UNICODE[21554] := 16#C156;
   // GBK_TO_UNICODE[21555] := 16#7F7A;
   // GBK_TO_UNICODE[21556] := 16#C157;
   // GBK_TO_UNICODE[21557] := 16#7F7B;
   // GBK_TO_UNICODE[21558] := 16#C158;
   // GBK_TO_UNICODE[21559] := 16#7F7C;
   // GBK_TO_UNICODE[21560] := 16#C159;
   // GBK_TO_UNICODE[21561] := 16#7F7D;
   // GBK_TO_UNICODE[21562] := 16#C15A;
   // GBK_TO_UNICODE[21563] := 16#7F7F;
   // GBK_TO_UNICODE[21564] := 16#C15B;
   // GBK_TO_UNICODE[21565] := 16#7F80;
   // GBK_TO_UNICODE[21566] := 16#C15C;
   // GBK_TO_UNICODE[21567] := 16#7F82;
   // GBK_TO_UNICODE[21568] := 16#C15D;
   // GBK_TO_UNICODE[21569] := 16#7F83;
   // GBK_TO_UNICODE[21570] := 16#C15E;
   // GBK_TO_UNICODE[21571] := 16#7F84;
   // GBK_TO_UNICODE[21572] := 16#C15F;
   // GBK_TO_UNICODE[21573] := 16#7F85;
   // GBK_TO_UNICODE[21574] := 16#C160;
   // GBK_TO_UNICODE[21575] := 16#7F86;
   // GBK_TO_UNICODE[21576] := 16#C161;
   // GBK_TO_UNICODE[21577] := 16#7F87;
   // GBK_TO_UNICODE[21578] := 16#C162;
   // GBK_TO_UNICODE[21579] := 16#7F88;
   // GBK_TO_UNICODE[21580] := 16#C163;
   // GBK_TO_UNICODE[21581] := 16#7F89;
   // GBK_TO_UNICODE[21582] := 16#C164;
   // GBK_TO_UNICODE[21583] := 16#7F8B;
   // GBK_TO_UNICODE[21584] := 16#C165;
   // GBK_TO_UNICODE[21585] := 16#7F8D;
   // GBK_TO_UNICODE[21586] := 16#C166;
   // GBK_TO_UNICODE[21587] := 16#7F8F;
   // GBK_TO_UNICODE[21588] := 16#C167;
   // GBK_TO_UNICODE[21589] := 16#7F90;
   // GBK_TO_UNICODE[21590] := 16#C168;
   // GBK_TO_UNICODE[21591] := 16#7F91;
   // GBK_TO_UNICODE[21592] := 16#C169;
   // GBK_TO_UNICODE[21593] := 16#7F92;
   // GBK_TO_UNICODE[21594] := 16#C16A;
   // GBK_TO_UNICODE[21595] := 16#7F93;
   // GBK_TO_UNICODE[21596] := 16#C16B;
   // GBK_TO_UNICODE[21597] := 16#7F95;
   // GBK_TO_UNICODE[21598] := 16#C16C;
   // GBK_TO_UNICODE[21599] := 16#7F96;
   // GBK_TO_UNICODE[21600] := 16#C16D;
   // GBK_TO_UNICODE[21601] := 16#7F97;
   // GBK_TO_UNICODE[21602] := 16#C16E;
   // GBK_TO_UNICODE[21603] := 16#7F98;
   // GBK_TO_UNICODE[21604] := 16#C16F;
   // GBK_TO_UNICODE[21605] := 16#7F99;
   // GBK_TO_UNICODE[21606] := 16#C170;
   // GBK_TO_UNICODE[21607] := 16#7F9B;
   // GBK_TO_UNICODE[21608] := 16#C171;
   // GBK_TO_UNICODE[21609] := 16#7F9C;
   // GBK_TO_UNICODE[21610] := 16#C172;
   // GBK_TO_UNICODE[21611] := 16#7FA0;
   // GBK_TO_UNICODE[21612] := 16#C173;
   // GBK_TO_UNICODE[21613] := 16#7FA2;
   // GBK_TO_UNICODE[21614] := 16#C174;
   // GBK_TO_UNICODE[21615] := 16#7FA3;
   // GBK_TO_UNICODE[21616] := 16#C175;
   // GBK_TO_UNICODE[21617] := 16#7FA5;
   // GBK_TO_UNICODE[21618] := 16#C176;
   // GBK_TO_UNICODE[21619] := 16#7FA6;
   // GBK_TO_UNICODE[21620] := 16#C177;
   // GBK_TO_UNICODE[21621] := 16#7FA8;
   // GBK_TO_UNICODE[21622] := 16#C178;
   // GBK_TO_UNICODE[21623] := 16#7FA9;
   // GBK_TO_UNICODE[21624] := 16#C179;
   // GBK_TO_UNICODE[21625] := 16#7FAA;
   // GBK_TO_UNICODE[21626] := 16#C17A;
   // GBK_TO_UNICODE[21627] := 16#7FAB;
   // GBK_TO_UNICODE[21628] := 16#C17B;
   // GBK_TO_UNICODE[21629] := 16#7FAC;
   // GBK_TO_UNICODE[21630] := 16#C17C;
   // GBK_TO_UNICODE[21631] := 16#7FAD;
   // GBK_TO_UNICODE[21632] := 16#C17D;
   // GBK_TO_UNICODE[21633] := 16#7FAE;
   // GBK_TO_UNICODE[21634] := 16#C17E;
   // GBK_TO_UNICODE[21635] := 16#7FB1;
   // GBK_TO_UNICODE[21636] := 16#C180;
   // GBK_TO_UNICODE[21637] := 16#7FB3;
   // GBK_TO_UNICODE[21638] := 16#C181;
   // GBK_TO_UNICODE[21639] := 16#7FB4;
   // GBK_TO_UNICODE[21640] := 16#C182;
   // GBK_TO_UNICODE[21641] := 16#7FB5;
   // GBK_TO_UNICODE[21642] := 16#C183;
   // GBK_TO_UNICODE[21643] := 16#7FB6;
   // GBK_TO_UNICODE[21644] := 16#C184;
   // GBK_TO_UNICODE[21645] := 16#7FB7;
   // GBK_TO_UNICODE[21646] := 16#C185;
   // GBK_TO_UNICODE[21647] := 16#7FBA;
   // GBK_TO_UNICODE[21648] := 16#C186;
   // GBK_TO_UNICODE[21649] := 16#7FBB;
   // GBK_TO_UNICODE[21650] := 16#C187;
   // GBK_TO_UNICODE[21651] := 16#7FBE;
   // GBK_TO_UNICODE[21652] := 16#C188;
   // GBK_TO_UNICODE[21653] := 16#7FC0;
   // GBK_TO_UNICODE[21654] := 16#C189;
   // GBK_TO_UNICODE[21655] := 16#7FC2;
   // GBK_TO_UNICODE[21656] := 16#C18A;
   // GBK_TO_UNICODE[21657] := 16#7FC3;
   // GBK_TO_UNICODE[21658] := 16#C18B;
   // GBK_TO_UNICODE[21659] := 16#7FC4;
   // GBK_TO_UNICODE[21660] := 16#C18C;
   // GBK_TO_UNICODE[21661] := 16#7FC6;
   // GBK_TO_UNICODE[21662] := 16#C18D;
   // GBK_TO_UNICODE[21663] := 16#7FC7;
   // GBK_TO_UNICODE[21664] := 16#C18E;
   // GBK_TO_UNICODE[21665] := 16#7FC8;
   // GBK_TO_UNICODE[21666] := 16#C18F;
   // GBK_TO_UNICODE[21667] := 16#7FC9;
   // GBK_TO_UNICODE[21668] := 16#C190;
   // GBK_TO_UNICODE[21669] := 16#7FCB;
   // GBK_TO_UNICODE[21670] := 16#C191;
   // GBK_TO_UNICODE[21671] := 16#7FCD;
   // GBK_TO_UNICODE[21672] := 16#C192;
   // GBK_TO_UNICODE[21673] := 16#7FCF;
   // GBK_TO_UNICODE[21674] := 16#C193;
   // GBK_TO_UNICODE[21675] := 16#7FD0;
   // GBK_TO_UNICODE[21676] := 16#C194;
   // GBK_TO_UNICODE[21677] := 16#7FD1;
   // GBK_TO_UNICODE[21678] := 16#C195;
   // GBK_TO_UNICODE[21679] := 16#7FD2;
   // GBK_TO_UNICODE[21680] := 16#C196;
   // GBK_TO_UNICODE[21681] := 16#7FD3;
   // GBK_TO_UNICODE[21682] := 16#C197;
   // GBK_TO_UNICODE[21683] := 16#7FD6;
   // GBK_TO_UNICODE[21684] := 16#C198;
   // GBK_TO_UNICODE[21685] := 16#7FD7;
   // GBK_TO_UNICODE[21686] := 16#C199;
   // GBK_TO_UNICODE[21687] := 16#7FD9;
   // GBK_TO_UNICODE[21688] := 16#C19A;
   // GBK_TO_UNICODE[21689] := 16#7FDA;
   // GBK_TO_UNICODE[21690] := 16#C19B;
   // GBK_TO_UNICODE[21691] := 16#7FDB;
   // GBK_TO_UNICODE[21692] := 16#C19C;
   // GBK_TO_UNICODE[21693] := 16#7FDC;
   // GBK_TO_UNICODE[21694] := 16#C19D;
   // GBK_TO_UNICODE[21695] := 16#7FDD;
   // GBK_TO_UNICODE[21696] := 16#C19E;
   // GBK_TO_UNICODE[21697] := 16#7FDE;
   // GBK_TO_UNICODE[21698] := 16#C19F;
   // GBK_TO_UNICODE[21699] := 16#7FE2;
   // GBK_TO_UNICODE[21700] := 16#C1A0;
   // GBK_TO_UNICODE[21701] := 16#7FE3;
   // GBK_TO_UNICODE[21702] := 16#C1A1;
   // GBK_TO_UNICODE[21703] := 16#75E2;
   // GBK_TO_UNICODE[21704] := 16#C1A2;
   // GBK_TO_UNICODE[21705] := 16#7ACB;
   // GBK_TO_UNICODE[21706] := 16#C1A3;
   // GBK_TO_UNICODE[21707] := 16#7C92;
   // GBK_TO_UNICODE[21708] := 16#C1A4;
   // GBK_TO_UNICODE[21709] := 16#6CA5;
   // GBK_TO_UNICODE[21710] := 16#C1A5;
   // GBK_TO_UNICODE[21711] := 16#96B6;
   // GBK_TO_UNICODE[21712] := 16#C1A6;
   // GBK_TO_UNICODE[21713] := 16#529B;
   // GBK_TO_UNICODE[21714] := 16#C1A7;
   // GBK_TO_UNICODE[21715] := 16#7483;
   // GBK_TO_UNICODE[21716] := 16#C1A8;
   // GBK_TO_UNICODE[21717] := 16#54E9;
   // GBK_TO_UNICODE[21718] := 16#C1A9;
   // GBK_TO_UNICODE[21719] := 16#4FE9;
   // GBK_TO_UNICODE[21720] := 16#C1AA;
   // GBK_TO_UNICODE[21721] := 16#8054;
   // GBK_TO_UNICODE[21722] := 16#C1AB;
   // GBK_TO_UNICODE[21723] := 16#83B2;
   // GBK_TO_UNICODE[21724] := 16#C1AC;
   // GBK_TO_UNICODE[21725] := 16#8FDE;
   // GBK_TO_UNICODE[21726] := 16#C1AD;
   // GBK_TO_UNICODE[21727] := 16#9570;
   // GBK_TO_UNICODE[21728] := 16#C1AE;
   // GBK_TO_UNICODE[21729] := 16#5EC9;
   // GBK_TO_UNICODE[21730] := 16#C1AF;
   // GBK_TO_UNICODE[21731] := 16#601C;
   // GBK_TO_UNICODE[21732] := 16#C1B0;
   // GBK_TO_UNICODE[21733] := 16#6D9F;
   // GBK_TO_UNICODE[21734] := 16#C1B1;
   // GBK_TO_UNICODE[21735] := 16#5E18;
   // GBK_TO_UNICODE[21736] := 16#C1B2;
   // GBK_TO_UNICODE[21737] := 16#655B;
   // GBK_TO_UNICODE[21738] := 16#C1B3;
   // GBK_TO_UNICODE[21739] := 16#8138;
   // GBK_TO_UNICODE[21740] := 16#C1B4;
   // GBK_TO_UNICODE[21741] := 16#94FE;
   // GBK_TO_UNICODE[21742] := 16#C1B5;
   // GBK_TO_UNICODE[21743] := 16#604B;
   // GBK_TO_UNICODE[21744] := 16#C1B6;
   // GBK_TO_UNICODE[21745] := 16#70BC;
   // GBK_TO_UNICODE[21746] := 16#C1B7;
   // GBK_TO_UNICODE[21747] := 16#7EC3;
   // GBK_TO_UNICODE[21748] := 16#C1B8;
   // GBK_TO_UNICODE[21749] := 16#7CAE;
   // GBK_TO_UNICODE[21750] := 16#C1B9;
   // GBK_TO_UNICODE[21751] := 16#51C9;
   // GBK_TO_UNICODE[21752] := 16#C1BA;
   // GBK_TO_UNICODE[21753] := 16#6881;
   // GBK_TO_UNICODE[21754] := 16#C1BB;
   // GBK_TO_UNICODE[21755] := 16#7CB1;
   // GBK_TO_UNICODE[21756] := 16#C1BC;
   // GBK_TO_UNICODE[21757] := 16#826F;
   // GBK_TO_UNICODE[21758] := 16#C1BD;
   // GBK_TO_UNICODE[21759] := 16#4E24;
   // GBK_TO_UNICODE[21760] := 16#C1BE;
   // GBK_TO_UNICODE[21761] := 16#8F86;
   // GBK_TO_UNICODE[21762] := 16#C1BF;
   // GBK_TO_UNICODE[21763] := 16#91CF;
   // GBK_TO_UNICODE[21764] := 16#C1C0;
   // GBK_TO_UNICODE[21765] := 16#667E;
   // GBK_TO_UNICODE[21766] := 16#C1C1;
   // GBK_TO_UNICODE[21767] := 16#4EAE;
   // GBK_TO_UNICODE[21768] := 16#C1C2;
   // GBK_TO_UNICODE[21769] := 16#8C05;
   // GBK_TO_UNICODE[21770] := 16#C1C3;
   // GBK_TO_UNICODE[21771] := 16#64A9;
   // GBK_TO_UNICODE[21772] := 16#C1C4;
   // GBK_TO_UNICODE[21773] := 16#804A;
   // GBK_TO_UNICODE[21774] := 16#C1C5;
   // GBK_TO_UNICODE[21775] := 16#50DA;
   // GBK_TO_UNICODE[21776] := 16#C1C6;
   // GBK_TO_UNICODE[21777] := 16#7597;
   // GBK_TO_UNICODE[21778] := 16#C1C7;
   // GBK_TO_UNICODE[21779] := 16#71CE;
   // GBK_TO_UNICODE[21780] := 16#C1C8;
   // GBK_TO_UNICODE[21781] := 16#5BE5;
   // GBK_TO_UNICODE[21782] := 16#C1C9;
   // GBK_TO_UNICODE[21783] := 16#8FBD;
   // GBK_TO_UNICODE[21784] := 16#C1CA;
   // GBK_TO_UNICODE[21785] := 16#6F66;
   // GBK_TO_UNICODE[21786] := 16#C1CB;
   // GBK_TO_UNICODE[21787] := 16#4E86;
   // GBK_TO_UNICODE[21788] := 16#C1CC;
   // GBK_TO_UNICODE[21789] := 16#6482;
   // GBK_TO_UNICODE[21790] := 16#C1CD;
   // GBK_TO_UNICODE[21791] := 16#9563;
   // GBK_TO_UNICODE[21792] := 16#C1CE;
   // GBK_TO_UNICODE[21793] := 16#5ED6;
   // GBK_TO_UNICODE[21794] := 16#C1CF;
   // GBK_TO_UNICODE[21795] := 16#6599;
   // GBK_TO_UNICODE[21796] := 16#C1D0;
   // GBK_TO_UNICODE[21797] := 16#5217;
   // GBK_TO_UNICODE[21798] := 16#C1D1;
   // GBK_TO_UNICODE[21799] := 16#88C2;
   // GBK_TO_UNICODE[21800] := 16#C1D2;
   // GBK_TO_UNICODE[21801] := 16#70C8;
   // GBK_TO_UNICODE[21802] := 16#C1D3;
   // GBK_TO_UNICODE[21803] := 16#52A3;
   // GBK_TO_UNICODE[21804] := 16#C1D4;
   // GBK_TO_UNICODE[21805] := 16#730E;
   // GBK_TO_UNICODE[21806] := 16#C1D5;
   // GBK_TO_UNICODE[21807] := 16#7433;
   // GBK_TO_UNICODE[21808] := 16#C1D6;
   // GBK_TO_UNICODE[21809] := 16#6797;
   // GBK_TO_UNICODE[21810] := 16#C1D7;
   // GBK_TO_UNICODE[21811] := 16#78F7;
   // GBK_TO_UNICODE[21812] := 16#C1D8;
   // GBK_TO_UNICODE[21813] := 16#9716;
   // GBK_TO_UNICODE[21814] := 16#C1D9;
   // GBK_TO_UNICODE[21815] := 16#4E34;
   // GBK_TO_UNICODE[21816] := 16#C1DA;
   // GBK_TO_UNICODE[21817] := 16#90BB;
   // GBK_TO_UNICODE[21818] := 16#C1DB;
   // GBK_TO_UNICODE[21819] := 16#9CDE;
   // GBK_TO_UNICODE[21820] := 16#C1DC;
   // GBK_TO_UNICODE[21821] := 16#6DCB;
   // GBK_TO_UNICODE[21822] := 16#C1DD;
   // GBK_TO_UNICODE[21823] := 16#51DB;
   // GBK_TO_UNICODE[21824] := 16#C1DE;
   // GBK_TO_UNICODE[21825] := 16#8D41;
   // GBK_TO_UNICODE[21826] := 16#C1DF;
   // GBK_TO_UNICODE[21827] := 16#541D;
   // GBK_TO_UNICODE[21828] := 16#C1E0;
   // GBK_TO_UNICODE[21829] := 16#62CE;
   // GBK_TO_UNICODE[21830] := 16#C1E1;
   // GBK_TO_UNICODE[21831] := 16#73B2;
   // GBK_TO_UNICODE[21832] := 16#C1E2;
   // GBK_TO_UNICODE[21833] := 16#83F1;
   // GBK_TO_UNICODE[21834] := 16#C1E3;
   // GBK_TO_UNICODE[21835] := 16#96F6;
   // GBK_TO_UNICODE[21836] := 16#C1E4;
   // GBK_TO_UNICODE[21837] := 16#9F84;
   // GBK_TO_UNICODE[21838] := 16#C1E5;
   // GBK_TO_UNICODE[21839] := 16#94C3;
   // GBK_TO_UNICODE[21840] := 16#C1E6;
   // GBK_TO_UNICODE[21841] := 16#4F36;
   // GBK_TO_UNICODE[21842] := 16#C1E7;
   // GBK_TO_UNICODE[21843] := 16#7F9A;
   // GBK_TO_UNICODE[21844] := 16#C1E8;
   // GBK_TO_UNICODE[21845] := 16#51CC;
   // GBK_TO_UNICODE[21846] := 16#C1E9;
   // GBK_TO_UNICODE[21847] := 16#7075;
   // GBK_TO_UNICODE[21848] := 16#C1EA;
   // GBK_TO_UNICODE[21849] := 16#9675;
   // GBK_TO_UNICODE[21850] := 16#C1EB;
   // GBK_TO_UNICODE[21851] := 16#5CAD;
   // GBK_TO_UNICODE[21852] := 16#C1EC;
   // GBK_TO_UNICODE[21853] := 16#9886;
   // GBK_TO_UNICODE[21854] := 16#C1ED;
   // GBK_TO_UNICODE[21855] := 16#53E6;
   // GBK_TO_UNICODE[21856] := 16#C1EE;
   // GBK_TO_UNICODE[21857] := 16#4EE4;
   // GBK_TO_UNICODE[21858] := 16#C1EF;
   // GBK_TO_UNICODE[21859] := 16#6E9C;
   // GBK_TO_UNICODE[21860] := 16#C1F0;
   // GBK_TO_UNICODE[21861] := 16#7409;
   // GBK_TO_UNICODE[21862] := 16#C1F1;
   // GBK_TO_UNICODE[21863] := 16#69B4;
   // GBK_TO_UNICODE[21864] := 16#C1F2;
   // GBK_TO_UNICODE[21865] := 16#786B;
   // GBK_TO_UNICODE[21866] := 16#C1F3;
   // GBK_TO_UNICODE[21867] := 16#998F;
   // GBK_TO_UNICODE[21868] := 16#C1F4;
   // GBK_TO_UNICODE[21869] := 16#7559;
   // GBK_TO_UNICODE[21870] := 16#C1F5;
   // GBK_TO_UNICODE[21871] := 16#5218;
   // GBK_TO_UNICODE[21872] := 16#C1F6;
   // GBK_TO_UNICODE[21873] := 16#7624;
   // GBK_TO_UNICODE[21874] := 16#C1F7;
   // GBK_TO_UNICODE[21875] := 16#6D41;
   // GBK_TO_UNICODE[21876] := 16#C1F8;
   // GBK_TO_UNICODE[21877] := 16#67F3;
   // GBK_TO_UNICODE[21878] := 16#C1F9;
   // GBK_TO_UNICODE[21879] := 16#516D;
   // GBK_TO_UNICODE[21880] := 16#C1FA;
   // GBK_TO_UNICODE[21881] := 16#9F99;
   // GBK_TO_UNICODE[21882] := 16#C1FB;
   // GBK_TO_UNICODE[21883] := 16#804B;
   // GBK_TO_UNICODE[21884] := 16#C1FC;
   // GBK_TO_UNICODE[21885] := 16#5499;
   // GBK_TO_UNICODE[21886] := 16#C1FD;
   // GBK_TO_UNICODE[21887] := 16#7B3C;
   // GBK_TO_UNICODE[21888] := 16#C1FE;
   // GBK_TO_UNICODE[21889] := 16#7ABF;
   // GBK_TO_UNICODE[21890] := 16#C240;
   // GBK_TO_UNICODE[21891] := 16#7FE4;
   // GBK_TO_UNICODE[21892] := 16#C241;
   // GBK_TO_UNICODE[21893] := 16#7FE7;
   // GBK_TO_UNICODE[21894] := 16#C242;
   // GBK_TO_UNICODE[21895] := 16#7FE8;
   // GBK_TO_UNICODE[21896] := 16#C243;
   // GBK_TO_UNICODE[21897] := 16#7FEA;
   // GBK_TO_UNICODE[21898] := 16#C244;
   // GBK_TO_UNICODE[21899] := 16#7FEB;
   // GBK_TO_UNICODE[21900] := 16#C245;
   // GBK_TO_UNICODE[21901] := 16#7FEC;
   // GBK_TO_UNICODE[21902] := 16#C246;
   // GBK_TO_UNICODE[21903] := 16#7FED;
   // GBK_TO_UNICODE[21904] := 16#C247;
   // GBK_TO_UNICODE[21905] := 16#7FEF;
   // GBK_TO_UNICODE[21906] := 16#C248;
   // GBK_TO_UNICODE[21907] := 16#7FF2;
   // GBK_TO_UNICODE[21908] := 16#C249;
   // GBK_TO_UNICODE[21909] := 16#7FF4;
   // GBK_TO_UNICODE[21910] := 16#C24A;
   // GBK_TO_UNICODE[21911] := 16#7FF5;
   // GBK_TO_UNICODE[21912] := 16#C24B;
   // GBK_TO_UNICODE[21913] := 16#7FF6;
   // GBK_TO_UNICODE[21914] := 16#C24C;
   // GBK_TO_UNICODE[21915] := 16#7FF7;
   // GBK_TO_UNICODE[21916] := 16#C24D;
   // GBK_TO_UNICODE[21917] := 16#7FF8;
   // GBK_TO_UNICODE[21918] := 16#C24E;
   // GBK_TO_UNICODE[21919] := 16#7FF9;
   // GBK_TO_UNICODE[21920] := 16#C24F;
   // GBK_TO_UNICODE[21921] := 16#7FFA;
   // GBK_TO_UNICODE[21922] := 16#C250;
   // GBK_TO_UNICODE[21923] := 16#7FFD;
   // GBK_TO_UNICODE[21924] := 16#C251;
   // GBK_TO_UNICODE[21925] := 16#7FFE;
   // GBK_TO_UNICODE[21926] := 16#C252;
   // GBK_TO_UNICODE[21927] := 16#7FFF;
   // GBK_TO_UNICODE[21928] := 16#C253;
   // GBK_TO_UNICODE[21929] := 16#8002;
   // GBK_TO_UNICODE[21930] := 16#C254;
   // GBK_TO_UNICODE[21931] := 16#8007;
   // GBK_TO_UNICODE[21932] := 16#C255;
   // GBK_TO_UNICODE[21933] := 16#8008;
   // GBK_TO_UNICODE[21934] := 16#C256;
   // GBK_TO_UNICODE[21935] := 16#8009;
   // GBK_TO_UNICODE[21936] := 16#C257;
   // GBK_TO_UNICODE[21937] := 16#800A;
   // GBK_TO_UNICODE[21938] := 16#C258;
   // GBK_TO_UNICODE[21939] := 16#800E;
   // GBK_TO_UNICODE[21940] := 16#C259;
   // GBK_TO_UNICODE[21941] := 16#800F;
   // GBK_TO_UNICODE[21942] := 16#C25A;
   // GBK_TO_UNICODE[21943] := 16#8011;
   // GBK_TO_UNICODE[21944] := 16#C25B;
   // GBK_TO_UNICODE[21945] := 16#8013;
   // GBK_TO_UNICODE[21946] := 16#C25C;
   // GBK_TO_UNICODE[21947] := 16#801A;
   // GBK_TO_UNICODE[21948] := 16#C25D;
   // GBK_TO_UNICODE[21949] := 16#801B;
   // GBK_TO_UNICODE[21950] := 16#C25E;
   // GBK_TO_UNICODE[21951] := 16#801D;
   // GBK_TO_UNICODE[21952] := 16#C25F;
   // GBK_TO_UNICODE[21953] := 16#801E;
   // GBK_TO_UNICODE[21954] := 16#C260;
   // GBK_TO_UNICODE[21955] := 16#801F;
   // GBK_TO_UNICODE[21956] := 16#C261;
   // GBK_TO_UNICODE[21957] := 16#8021;
   // GBK_TO_UNICODE[21958] := 16#C262;
   // GBK_TO_UNICODE[21959] := 16#8023;
   // GBK_TO_UNICODE[21960] := 16#C263;
   // GBK_TO_UNICODE[21961] := 16#8024;
   // GBK_TO_UNICODE[21962] := 16#C264;
   // GBK_TO_UNICODE[21963] := 16#802B;
   // GBK_TO_UNICODE[21964] := 16#C265;
   // GBK_TO_UNICODE[21965] := 16#802C;
   // GBK_TO_UNICODE[21966] := 16#C266;
   // GBK_TO_UNICODE[21967] := 16#802D;
   // GBK_TO_UNICODE[21968] := 16#C267;
   // GBK_TO_UNICODE[21969] := 16#802E;
   // GBK_TO_UNICODE[21970] := 16#C268;
   // GBK_TO_UNICODE[21971] := 16#802F;
   // GBK_TO_UNICODE[21972] := 16#C269;
   // GBK_TO_UNICODE[21973] := 16#8030;
   // GBK_TO_UNICODE[21974] := 16#C26A;
   // GBK_TO_UNICODE[21975] := 16#8032;
   // GBK_TO_UNICODE[21976] := 16#C26B;
   // GBK_TO_UNICODE[21977] := 16#8034;
   // GBK_TO_UNICODE[21978] := 16#C26C;
   // GBK_TO_UNICODE[21979] := 16#8039;
   // GBK_TO_UNICODE[21980] := 16#C26D;
   // GBK_TO_UNICODE[21981] := 16#803A;
   // GBK_TO_UNICODE[21982] := 16#C26E;
   // GBK_TO_UNICODE[21983] := 16#803C;
   // GBK_TO_UNICODE[21984] := 16#C26F;
   // GBK_TO_UNICODE[21985] := 16#803E;
   // GBK_TO_UNICODE[21986] := 16#C270;
   // GBK_TO_UNICODE[21987] := 16#8040;
   // GBK_TO_UNICODE[21988] := 16#C271;
   // GBK_TO_UNICODE[21989] := 16#8041;
   // GBK_TO_UNICODE[21990] := 16#C272;
   // GBK_TO_UNICODE[21991] := 16#8044;
   // GBK_TO_UNICODE[21992] := 16#C273;
   // GBK_TO_UNICODE[21993] := 16#8045;
   // GBK_TO_UNICODE[21994] := 16#C274;
   // GBK_TO_UNICODE[21995] := 16#8047;
   // GBK_TO_UNICODE[21996] := 16#C275;
   // GBK_TO_UNICODE[21997] := 16#8048;
   // GBK_TO_UNICODE[21998] := 16#C276;
   // GBK_TO_UNICODE[21999] := 16#8049;
   // GBK_TO_UNICODE[22000] := 16#C277;
   // GBK_TO_UNICODE[22001] := 16#804E;
   // GBK_TO_UNICODE[22002] := 16#C278;
   // GBK_TO_UNICODE[22003] := 16#804F;
   // GBK_TO_UNICODE[22004] := 16#C279;
   // GBK_TO_UNICODE[22005] := 16#8050;
   // GBK_TO_UNICODE[22006] := 16#C27A;
   // GBK_TO_UNICODE[22007] := 16#8051;
   // GBK_TO_UNICODE[22008] := 16#C27B;
   // GBK_TO_UNICODE[22009] := 16#8053;
   // GBK_TO_UNICODE[22010] := 16#C27C;
   // GBK_TO_UNICODE[22011] := 16#8055;
   // GBK_TO_UNICODE[22012] := 16#C27D;
   // GBK_TO_UNICODE[22013] := 16#8056;
   // GBK_TO_UNICODE[22014] := 16#C27E;
   // GBK_TO_UNICODE[22015] := 16#8057;
   // GBK_TO_UNICODE[22016] := 16#C280;
   // GBK_TO_UNICODE[22017] := 16#8059;
   // GBK_TO_UNICODE[22018] := 16#C281;
   // GBK_TO_UNICODE[22019] := 16#805B;
   // GBK_TO_UNICODE[22020] := 16#C282;
   // GBK_TO_UNICODE[22021] := 16#805C;
   // GBK_TO_UNICODE[22022] := 16#C283;
   // GBK_TO_UNICODE[22023] := 16#805D;
   // GBK_TO_UNICODE[22024] := 16#C284;
   // GBK_TO_UNICODE[22025] := 16#805E;
   // GBK_TO_UNICODE[22026] := 16#C285;
   // GBK_TO_UNICODE[22027] := 16#805F;
   // GBK_TO_UNICODE[22028] := 16#C286;
   // GBK_TO_UNICODE[22029] := 16#8060;
   // GBK_TO_UNICODE[22030] := 16#C287;
   // GBK_TO_UNICODE[22031] := 16#8061;
   // GBK_TO_UNICODE[22032] := 16#C288;
   // GBK_TO_UNICODE[22033] := 16#8062;
   // GBK_TO_UNICODE[22034] := 16#C289;
   // GBK_TO_UNICODE[22035] := 16#8063;
   // GBK_TO_UNICODE[22036] := 16#C28A;
   // GBK_TO_UNICODE[22037] := 16#8064;
   // GBK_TO_UNICODE[22038] := 16#C28B;
   // GBK_TO_UNICODE[22039] := 16#8065;
   // GBK_TO_UNICODE[22040] := 16#C28C;
   // GBK_TO_UNICODE[22041] := 16#8066;
   // GBK_TO_UNICODE[22042] := 16#C28D;
   // GBK_TO_UNICODE[22043] := 16#8067;
   // GBK_TO_UNICODE[22044] := 16#C28E;
   // GBK_TO_UNICODE[22045] := 16#8068;
   // GBK_TO_UNICODE[22046] := 16#C28F;
   // GBK_TO_UNICODE[22047] := 16#806B;
   // GBK_TO_UNICODE[22048] := 16#C290;
   // GBK_TO_UNICODE[22049] := 16#806C;
   // GBK_TO_UNICODE[22050] := 16#C291;
   // GBK_TO_UNICODE[22051] := 16#806D;
   // GBK_TO_UNICODE[22052] := 16#C292;
   // GBK_TO_UNICODE[22053] := 16#806E;
   // GBK_TO_UNICODE[22054] := 16#C293;
   // GBK_TO_UNICODE[22055] := 16#806F;
   // GBK_TO_UNICODE[22056] := 16#C294;
   // GBK_TO_UNICODE[22057] := 16#8070;
   // GBK_TO_UNICODE[22058] := 16#C295;
   // GBK_TO_UNICODE[22059] := 16#8072;
   // GBK_TO_UNICODE[22060] := 16#C296;
   // GBK_TO_UNICODE[22061] := 16#8073;
   // GBK_TO_UNICODE[22062] := 16#C297;
   // GBK_TO_UNICODE[22063] := 16#8074;
   // GBK_TO_UNICODE[22064] := 16#C298;
   // GBK_TO_UNICODE[22065] := 16#8075;
   // GBK_TO_UNICODE[22066] := 16#C299;
   // GBK_TO_UNICODE[22067] := 16#8076;
